# B&R Automation Studio project A65
Automation Studio 4.10.2.37

## Configuration Config1

CPU X20CP1382, AutomationRuntime D4.83, Build 4.1.2

### Task classes (Cpu.sw)
```
Cyclic#1 (cycle 2000 us, tolerance 2000 us):
  TaskFast <- Kontrol.TaskFast.TaskFast.prg
  FastMeter <- (binary)
  Program <- (binary)
  SslClient <- (binary)
  Server <- (binary)
  Client <- (binary)
  QDTA_IO <- (binary)
Cyclic#2 (cycle 10000 us, tolerance 10000 us):
  Protection <- Kontrol.Protection.Protection.prg
  Control <- Kontrol.Control.Control.prg
Cyclic#3 (cycle 100000 us, tolerance 100000 us):
  WatchDog <- WatchDog.WatchDog.prg
  System <- Kontrol.System.System.prg
  Hardware <- Kontrol.Hardware.Hardware.prg
  ProtUpdate <- Kontrol.Protection.ProtUpdate.prg
  Command <- Kontrol.Command.Command.prg
  cb52 <- Kontrol.CB52.cb52.prg
Cyclic#4 (cycle 200000 us, tolerance 200000 us):
  Auto <- Auto.Auto.prg
Cyclic#6 (cycle 50000 us, tolerance 3000000 us):
  MDB_Comand <- Auto.Modbus.MDB_Comando.prg
  MDB_Status <- Auto.Modbus.MDB_Status.prg
  MDB_Alarme <- Auto.Modbus.MDB_Alarme.prg
  MDB_Medida <- Auto.Modbus.MDB_Medida.prg
  MDB_Parame <- Auto.Modbus.MDB_Parametro.prg
Cyclic#7 (cycle 20000 us, tolerance 10000000 us):
  Event <- Kontrol.Event.Event.prg
  Comm <- Comm.Comm.prg
Cyclic#8 (cycle 50000 us, tolerance 10000000 us):
  File <- Kontrol.File.File.prg
Binaries: TCData, udbdef, ashwd, sysconf, asfw, arconfig, iomap, Role, User, ashwac, OpcUaMap, vccddbox, ihm01, ihm02, ihm03, vccpopup, vcpfx20, vcctrend, vccstr, vcmgr, vcpdsw, vcpdvnc, vccline, vccovl, arial, vcdsint, vccnum, vcalarm, vctcal, vccbtn, vcnet, vccbmp, vcrt, vcshared, vccdt, vcgclass, vcfntttf, vcbclass, vcdsloc, vcfile, arialbd, vcctext, vccshape, vccgauge, vcpkat, 10111548$f, Visu02, Visu03, Visu01, vccbar, vccslider, vcchspot, vccurl, vccalarm, vcchtml, vcxml
Libraries: operator, runtime, LoopConR, sys_lib, brsystem, AsTCP, AsIecCon, astime, AsBrStr, AsARCfg, AsXml, FileIO, AsIOAcc, standard, AsSem, IecCheck, DRV_mbus, dvframe, DataObj, Pgs0985, PgsAI4622, PgsAO4622, PgsAuto, PgsCfgNet, PgsComm, PgsControl, PgsEvent, PgsFileSys, PgsProt, PgsTag, PgsTagLink, PgsTelnet, vcresman, ashw
```

### Hardware
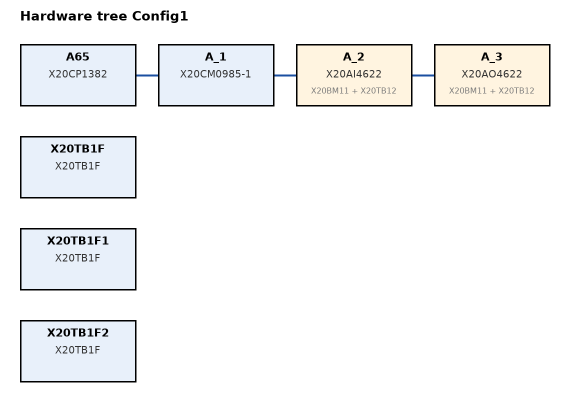
```
A65 : X20CP1382 v1.11.0.0  [X1 -> X1.SL; X2 -> X2.SL; X3 -> X3.SL]
  Module X1 (Type=X1, Virtual=true, Version=1.11.0.0)
    Connection (Connector=SS1, TargetModule=X20TB1F, TargetConnector=SS)
    Connection (Connector=SL, TargetModule=A65, TargetConnector=X1)
    X1AI_ChannelType01 = PT1000
    X1AI_ChannelType02 = 4 to 20mA
    X1AI2_LowerLimit_420mA = -8192
  Module X2 (Type=X2, Virtual=true, Version=1.11.0.0)
    Connection (Connector=SS1, TargetModule=X20TB1F1, TargetConnector=SS)
    Connection (Connector=SL, TargetModule=A65, TargetConnector=X2)
    X2CounterFunction = Edge
    X2CounterTimeInfo = 32Bit
  Module X3 (Type=X3, Virtual=true, Version=1.11.0.0)
    Connection (Connector=SS1, TargetModule=X20TB1F2, TargetConnector=SS)
    Connection (Connector=SL, TargetModule=A65, TargetConnector=X3)
  Connector IF1:
    Baudrate = 19200
  Connector IF2:
    ActivateDevice = 1
    Mode = Manual
    InternetAddress = 192.168.0.100
    SubnetMask = 255.255.255.0
    InaNodeNumber = 1
    Vnc1
    VncKeyMappingFile1 = 
    VncRefreshRate1 = 250
    ActivateSnmp = 2
    ActivateModbus = 1
    NumSlaves = -1
    NumAllBlocks = -1
    MemSizeIn = -1
    MemSizeOut = -1
  Connector IF3:
    DNAConfiguration = manual
    ActivateIna = 1
  ConfigurationID = A65
  RemanentGlobalPvSize = 10940
  EnableUsbRemoteInstall = 1
  EnableCfRemoteInstall = 1
  SystemTick = 2000
  IdleTaskClass = 8
  TaskClassIdleTime = 4000
  Cyclic1Duration = 2000
  Cyclic1Tolerance = 2000
  Cyclic2Duration = 10000
  Cyclic2Tolerance = 10000
  Cyclic3Duration = 100000
  Cyclic3Tolerance = 100000
  Cyclic4Duration = 200000
  Cyclic4Tolerance = 200000
  Cyclic5Duration = 500000
  Cyclic5Tolerance = 500000
  Cyclic6Duration = 50000
  Cyclic6Tolerance = 3000000
  Cyclic7Duration = 20000
  Cyclic7Tolerance = 10000000
  Cyclic8Duration = 50000
  Cyclic8Tolerance = 10000000
  FileDevice1
  FileDeviceName1 = 
  FileDevicePath1 = 
  TimeZone = 105
  ActivateSntp = 1
  SntpcServAddr1 = a.st1.ntp.br
  SntpcServAddr2 = b.st1.ntp.br
  SntpcServAddr3 = c.st1.ntp.br
  SntpcServAddr4 = d.st1.ntp.br
  EthernetDefaultGateway = 192.168.0.1
  FtpUser1
  FtpUsername1 = progressul
  FtpUserPassword1 = vk2iY3J4UkERtYbEJrmZIzULlFJLyE0YoKo7iPp2s1I=
  FtpUserSalt1 = 6vig95Eg
  FTPAccessRight1 = 0
  FTPMSPartition1 = SYSTEM
  FTPMSpath1 = 
  ActivateOpcUa = 1
  OpcUaInformationModels_PV_Version = 1
A_1 : X20CM0985-1 v2.2.0.0  [X2X1 -> A65.IF6]
  Supervision = off
  ReadBack = on
  FuncDO5 = NetErrorUser
  Timestamps = on
  GenErrorReset = on
  GenErrorCheck = phaseline
  NetConfig = 3Phase
  SyncConfig = X4X3
A_2 : X20AI4622 v1.1.0.0  [SS1 -> X20TB12.SS; SL -> X20BM11.SL1]
  Supervision = off
  ChannelType01 = 4 to 20mA
  ChannelType02 = 4 to 20mA
  ChannelType03 = 4 to 20mA
  ChannelType04 = 4 to 20mA
A_3 : X20AO4622 v1.2.0.0  [SS1 -> X20TB12j.SS; SL -> X20BM11i.SL1]
  Supervision = off
  ChannelType01 = 0 to 20mA
  ChannelType02 = 4 to 20mA
  ChannelType03 = 4 to 20mA
  ChannelType04 = 4 to 20mA
X20BM11 : X20BM11 v1.0.0.1  [X2X1 -> A_1.X2X2]
X20BM11i : X20BM11 v1.0.0.1  [X2X1 -> X20BM11.X2X2]
X20TB12 : X20TB12 v1.0.0.0
X20TB12j : X20TB12 v1.0.0.0
X20TB1F : X20TB1F v1.0.0.0
X20TB1F1 : X20TB1F v1.0.0.0
X20TB1F2 : X20TB1F v1.0.0.0
```

### IoMap.iom - A65/IoMap.iom
```iecst
(*********************************************************************************
 * Copyright: Microsoft
 * Author:    sandrionir
 * Created:   February 21, 2017/7:19 AM
 *********************************************************************************
 * IO mapping
 *********************************************************************************)
VAR_CONFIG
	Cyclic#4.HW.TemperatureENV AT %IW."A65".TemperatureENV;
	Cyclic#4.HW.TemperatureCPU AT %IW."A65".TemperatureCPU;
	Cyclic#2.cm0985IO.di.T32N AT %IX."A_1".StatusInput32;
	Cyclic#2.cm0985IO.di.T32P AT %IX."A_1".StatusInput31;
	Cyclic#2.cm0985IO.di.T27_2 AT %IX."A_1".StatusInput18;
	Cyclic#2.cm0985IO.di.T32Q AT %IX."A_1".StatusInput10;
	Cyclic#2.cm0985IO.di.T51 AT %IX."A_1".StatusInput09;
	Cyclic#2.cm0985IO.di.T50 AT %IX."A_1".StatusInput08;
	Cyclic#2.cm0985IO.di.T50N AT %IX."A_1".StatusInput07;
	Cyclic#2.cm0985IO.di.T60I AT %IX."A_1".StatusInput06;
	Cyclic#2.cm0985IO.di.T60V AT %IX."A_1".StatusInput05;
	Cyclic#2.cm0985IO.di.T81U AT %IX."A_1".StatusInput04;
	Cyclic#2.cm0985IO.di.T81O AT %IX."A_1".StatusInput03;
	Cyclic#2.cm0985IO.di.T27_1 AT %IX."A_1".StatusInput02;
	Cyclic#2.cm0985IO.di.T59 AT %IX."A_1".StatusInput01;
	Cyclic#2.::cm0985IO.do.RstError AT %QX."A_1".ResetGeneratorErrors;
	Cyclic#2.HW.Modulos.A_1_OK AT %IX."A_1".ModuleOk;
	Cyclic#2.cm0985IO.do.INVDO05 AT %QX."A_1".InvertDO5;
	Cyclic#2.Protection.do.trip_86h AT %QX."A_1".DigitalOutput06;
	Cyclic#2.Protection.do.trip_86e AT %QX."A_1".DigitalOutput05;
	Cyclic#2.::cm0985IO.do.SyncDeadBus AT %QX."A_1".ConfigOutput19;
	Cyclic#2.::cm0985IO.do.SyncCheck AT %QX."A_1".ConfigOutput18;
	Cyclic#2.::cm0985IO.do.SyncSlip AT %QX."A_1".ConfigOutput17;
	Cyclic#2.cm0985Meter.Registers.AnalogInput43 AT %ID."A_1".AnalogInput43;
	Cyclic#2.cm0985Meter.Registers.AnalogInput42 AT %ID."A_1".AnalogInput42;
	Cyclic#2.cm0985Meter.Registers.AnalogInput41 AT %ID."A_1".AnalogInput41;
	Cyclic#2.cm0985Meter.Registers.AnalogInput40 AT %ID."A_1".AnalogInput40;
	Cyclic#2.cm0985Meter.Registers.AnalogInput39 AT %ID."A_1".AnalogInput39;
	Cyclic#2.cm0985Meter.Registers.AnalogInput38 AT %ID."A_1".AnalogInput38;
	Cyclic#2.cm0985Meter.Registers.AnalogInput35 AT %IW."A_1".AnalogInput35;
	Cyclic#2.cm0985Meter.Registers.AnalogInput30 AT %IW."A_1".AnalogInput30;
	Cyclic#2.cm0985Meter.Registers.AnalogInput29 AT %IW."A_1".AnalogInput29;
	Cyclic#2.cm0985Meter.Registers.AnalogInput27 AT %IW."A_1".AnalogInput27;
	Cyclic#2.cm0985Meter.Registers.AnalogInput26 AT %IW."A_1".AnalogInput26;
	Cyclic#2.cm0985Meter.Registers.AnalogInput25 AT %IW."A_1".AnalogInput25;
	Cyclic#2.cm0985Meter.Registers.AnalogInput24 AT %IW."A_1".AnalogInput24;
	Cyclic#2.cm0985Meter.Registers.AnalogInput23 AT %IW."A_1".AnalogInput23;
	Cyclic#2.cm0985Meter.Registers.AnalogInput22 AT %IW."A_1".AnalogInput22;
	Cyclic#2.cm0985Meter.Registers.AnalogInput21 AT %IW."A_1".AnalogInput21;
	Cyclic#2.cm0985Meter.Registers.AnalogInput20 AT %IW."A_1".AnalogInput20;
	Cyclic#2.cm0985Meter.Registers.AnalogInput19 AT %IW."A_1".AnalogInput19;
	Cyclic#2.cm0985Meter.Registers.AnalogInput18 AT %IW."A_1".AnalogInput18;
	Cyclic#2.cm0985Meter.Registers.AnalogInput17 AT %IW."A_1".AnalogInput17;
	Cyclic#2.cm0985Meter.Registers.AnalogInput16 AT %IW."A_1".AnalogInput16;
	Cyclic#2.cm0985Meter.Registers.AnalogInput15 AT %IW."A_1".AnalogInput15;
	Cyclic#2.cm0985Meter.Registers.AnalogInput14 AT %IW."A_1".AnalogInput14;
	Cyclic#2.cm0985Meter.Registers.AnalogInput13 AT %IW."A_1".AnalogInput13;
	Cyclic#2.cm0985Meter.Registers.AnalogInput12 AT %IW."A_1".AnalogInput12;
	Cyclic#2.cm0985Meter.Registers.AnalogInput11 AT %IW."A_1".AnalogInput11;
	Cyclic#2.cm0985Meter.Registers.AnalogInput10 AT %IW."A_1".AnalogInput10;
	Cyclic#2.cm0985Meter.Registers.AnalogInput09 AT %IW."A_1".AnalogInput09;
	Cyclic#2.cm0985Meter.Registers.AnalogInput08 AT %IW."A_1".AnalogInput08;
	Cyclic#2.cm0985Meter.Registers.AnalogInput07 AT %IW."A_1".AnalogInput07;
	Cyclic#2.cm0985Meter.Registers.AnalogInput06 AT %IW."A_1".AnalogInput06;
	Cyclic#2.cm0985Meter.Registers.AnalogInput05 AT %IW."A_1".AnalogInput05;
	Cyclic#2.cm0985Meter.Registers.AnalogInput04 AT %IW."A_1".AnalogInput04;
	Cyclic#2.cm0985Meter.Registers.AnalogInput03 AT %IW."A_1".AnalogInput03;
	Cyclic#2.cm0985Meter.Registers.AnalogInput02 AT %IW."A_1".AnalogInput02;
	Cyclic#2.cm0985Meter.Registers.AnalogInput01 AT %IW."A_1".AnalogInput01;
	Cyclic#5.Control:rpm1.MasterCount AT %ID."X2".Counter01Value;
	Cyclic#5.Control:rpm1.MasterTime AT %ID."X2".Counter01TimeChanged;
	Cyclic#2.cm0985IO.di.UgPhSeqFault AT %IX."A_1".StatusInput19;
	Cyclic#2.cm0985IO.di.IgPhSeqFault AT %IX."A_1".StatusInput20;
	Cyclic#2.cm0985IO.di.UbPhSeqFault AT %IX."A_1".StatusInput21;
	Cyclic#2.cm0985IO.di.Us1PhSeqFault AT %IX."A_1".StatusInput22;
	Cyclic#2.::cm0985IO.di.PS24VFault AT %IX."A_1".StatusInput16;
	Cyclic#4.HW.SerialNumber AT %ID."A65".SerialNumber;
	Cyclic#4.HW.ModuleID AT %IW."A65".ModuleID;
	Cyclic#5.Control:rpm2.MasterCount AT %ID."X2".Counter02Value;
	Cyclic#5.Control:rpm2.MasterTime AT %ID."X2".Counter02TimeChanged;
	Cyclic#2.cm0985Meter.Registers.AnalogInput33 AT %IW."A_1".AnalogInput33;
	Cyclic#2.cm0985Meter.Registers.AnalogInput34 AT %IW."A_1".AnalogInput34;
	Cyclic#2.cm0985Meter.Registers.AnalogInput31 AT %IW."A_1".AnalogInput31;
	Cyclic#2.cm0985Meter.Registers.AnalogInput32 AT %IW."A_1".AnalogInput32;
	HW.FalhaFonteIO AT %IX."X3".StatusInput01;
	Protection.ai.ExcTemp AT %IW."X1".AnalogInput01;
	A65.ai.if AT %IW."X1".AnalogInput02;
	A65.di.dead_bus_enable AT %IX."X2".DigitalInput05;
	A65.di.avr_enable AT %IX."X2".DigitalInput01;
	A65.di.avr_ctrl_qm_enable AT %IX."X2".DigitalInput02;
	A65.di.avr_ctrl_pf_enable AT %IX."X2".DigitalInput03;
	A65.di.sync_enable AT %IX."X2".DigitalInput04;
	CB52.di.closed AT %IX."X2".DigitalInput06;
	A65.di.remote AT %IX."X2".DigitalInput07;
	A65.di.gov_trip AT %IX."X2".DigitalInput08;
	A65.di.avr_trip AT %IX."X2".DigitalInput09;
	A65.di.reset AT %IX."X1".DigitalInput01;
	A65.di.gov_enable AT %IX."X1".DigitalInput02;
	A65.di.gov_ctrl_pwr_enable AT %IX."X1".DigitalInput03;
	A65.di.gov_unload AT %IX."X1".DigitalInput04;
	A65.do.watchdog AT %QX."X3".DigitalOutput01;
	A65.do.gov_on AT %QX."X3".DigitalOutput02;
	A65.do.power_zero AT %QX."X3".DigitalOutput03;
	A65.ao.pwr AT %QW."A_3".AnalogOutput01;
	A65.ao.pos1 AT %QW."A_3".AnalogOutput02;
	Cyclic#4.HW.Modulos.A_3_OK AT %IX."A_3".ModuleOk;
	HW.Modulos.X1_Status AT %IB."X1".StatusInput01;
	A65.ao.pos2 AT %QW."A_3".AnalogOutput03;
	A65.ao.pos3 AT %QW."A_3".AnalogOutput04;
	Protection.di.crowbar_ok AT %IX."X2".DigitalInput10;
	Protection.di.pwr_temp_ok AT %IX."X2".DigitalInput14;
	A65.do.rotation_zero AT %QX."X3".DigitalOutput04;
	A65.do.rotation_nominal AT %QX."X3".DigitalOutput05;
	A65.do.rotation_brake AT %QX."X3".DigitalOutput06;
	A65.do.avr_on AT %QX."X3".DigitalOutput07;
	A65.do.field_flash_on AT %QX."X3".DigitalOutput08;
	A65.do.voltage_nominal AT %QX."X3".DigitalOutput09;
	A65.do.sync_enabled AT %QX."X3".DigitalOutput10;
	A65.do.dead_bus_enabled AT %QX."X3".DigitalOutput11;
	Protection.do.trip_50bf AT %QX."X3".DigitalOutput12;
	HW.Modulos.A_2_OK AT %IX."A_2".ModuleOk;
	A65.ai.uf AT %IW."A_2".AnalogInput01;
	A65.ai.pos1 AT %IW."A_2".AnalogInput02;
	A65.ai.pos2 AT %IW."A_2".AnalogInput03;
	A65.ai.pos3 AT %IW."A_2".AnalogInput04;
END_VAR
```

## Logical view

Binary libraries used (declarations not repeated): AsARCfg, AsBrStr, AsIecCon, AsIOAcc, AsSem, AsTCP, astime, AsXml, brsystem, DataObj, DRV_mbus, dvframe, FileIO, LoopConR 4.10.0, operator, runtime, standard, sys_lib, IecCheck, Pgs0985 2.00.0, PgsAI4622, PgsAO4622, PgsCfgNet, PgsComm 1.10.1, PgsControl, PgsEvent 1.00.0, PgsFileSys, PgsProt 2.00.0, PgsTag 2.02.0, PgsTagLink, PgsTelnet 2.01.1, MDB_Comando

### Global.typ - Global data types
```iecst
(*********************************************************************************
 * Copyright: Microsoft
 * Author:    sandrionir
 * Created:   February 21, 2017/7:19 AM
 *********************************************************************************
 * Global data types of project
 *********************************************************************************)

TYPE
	PgsVersionType : 	STRUCT
		X : UINT;
		Y : UINT;
		Z : UINT;
	END_STRUCT;
	PgsHW : 	STRUCT
		TemperatureCPU : UINT;
		TemperatureENV : UINT;
		SerialNumber : UDINT;
		ModuleID : UINT;
		FalhaFonteIO : BOOL;
		Modulos : PgsHWModulos;
	END_STRUCT;
	PgsHWModulos : 	STRUCT
		X1_Status : USINT;
		A_1_OK : BOOL;
		A_2_OK : BOOL;
		A_3_OK : BOOL;
		A_4_OK : BOOL;
		A_5_OK : BOOL;
		A_6_OK : BOOL;
		A_7_OK : BOOL;
		A_8_OK : BOOL;
		A_9_OK : BOOL;
		A_10_OK : BOOL;
		A_11_OK : BOOL;
		A_12_OK : BOOL;
	END_STRUCT;
END_TYPE
```

### Global.var - Global variables
```iecst
(*********************************************************************************
 * Copyright: Microsoft
 * Author:    sandrionir
 * Created:   February 21, 2017/7:19 AM
 *********************************************************************************
 * Global variables of project
 *********************************************************************************)
VAR CONSTANT
	version : PgsVersionType := (X:=2,Y:=2,Z:=0);
END_VAR
(*Hardware*)
VAR
	HW : PgsHW;
END_VAR
```

### Package Logical/Libraries - Global libraries

### Library Logical/Libraries/Kontrol/PgsAuto (IEC)
Depends on: sys_lib

#### PgsAuto.fun - Exported functions and function blocks
```iecst
FUNCTION_BLOCK PgsEnergia
	VAR_INPUT
		enable : BOOL;
		reset : BOOL;
		power : REAL;
		set_inicial : BOOL;
		set_posEnergy : REAL;
		set_negEnergy : REAL;
	END_VAR
	VAR_OUTPUT
		posEnergy : LREAL;
		negEnergy : LREAL;
	END_VAR
	VAR
		priv : PgsEnergiaPrivType;
	END_VAR
END_FUNCTION_BLOCK

FUNCTION_BLOCK PgsHorimetro
	VAR_INPUT
		enable : BOOL;
		reset : BOOL;
		set_inicial : BOOL;
		set_total : REAL;
	END_VAR
	VAR_OUTPUT
		total : REAL;
		horas : REAL;
		minutos : REAL;
		segundos : REAL;
	END_VAR
	VAR
		priv : PgsHorimetroPrivType;
	END_VAR
END_FUNCTION_BLOCK

FUNCTION_BLOCK PgsManobra
	VAR_INPUT
		enable : BOOL;
		reset : BOOL;
		set_inicial : BOOL;
		set_total : REAL;
	END_VAR
	VAR_OUTPUT
		total : REAL;
	END_VAR
	VAR
		priv : PgsManobraPrivType;
	END_VAR
END_FUNCTION_BLOCK

FUNCTION PGS_MDB_TO_REAL : REAL (*TODO: Add your comment here*) (*$GROUP=User,$CAT=User,$GROUPICON=User.png,$CATICON=User.png*)
	VAR_INPUT
		IN : UDINT;
	END_VAR
	VAR
		pVar : REFERENCE TO REAL;
		varUint : ARRAY[0..1] OF UINT;
		varUint1 : REFERENCE TO ARRAY[0..1] OF UINT;
	END_VAR
END_FUNCTION

FUNCTION PGS_REAL_TO_MDB : UDINT (*TODO: Add your comment here*) (*$GROUP=User,$CAT=User,$GROUPICON=User.png,$CATICON=User.png*)
	VAR_INPUT
		IN : REAL;
	END_VAR
	VAR
		pVar : REFERENCE TO UDINT;
		varUint : ARRAY[0..1] OF UINT;
		varUint1 : REFERENCE TO ARRAY[0..1] OF UINT;
	END_VAR
END_FUNCTION

{REDUND_ERROR} FUNCTION PGS_MDB_TO_DINT : DINT (*TODO: Add your comment here*) (*$GROUP=User,$CAT=User,$GROUPICON=User.png,$CATICON=User.png*)
	VAR_INPUT
		HIGH : UINT;
		LOW : UINT;
	END_VAR
	VAR
		pVar : REFERENCE TO DINT;
		varUint : ARRAY[0..1] OF UINT;
	END_VAR
END_FUNCTION

{REDUND_ERROR} FUNCTION PGS_MDB_TO_UDINT : UDINT (*TODO: Add your comment here*) (*$GROUP=User,$CAT=User,$GROUPICON=User.png,$CATICON=User.png*)
	VAR_INPUT
		HIGH : UINT;
		LOW : UINT;
	END_VAR
	VAR
		pVar : REFERENCE TO UDINT;
		varUint : ARRAY[0..1] OF UINT;
	END_VAR
END_FUNCTION

FUNCTION_BLOCK PgsAlarme
	VAR_INPUT
		IN : BOOL; (*input signal*)
		PT : TIME; (*delay time*)
		RESET : BOOL; (*resets output Q1*)
	END_VAR
	VAR_OUTPUT
		Q : BOOL; (*rising edge of the input signal is delayed by PT*)
	END_VAR
	VAR
		ton : TON;
	END_VAR
END_FUNCTION_BLOCK

{REDUND_ERROR} FUNCTION_BLOCK PgsFiltro (*TODO: Add your comment here*) (*$GROUP=User,$CAT=User,$GROUPICON=User.png,$CATICON=User.png*)
	VAR_INPUT
		IN : {REDUND_UNREPLICABLE} REAL;
		CTE : {REDUND_UNREPLICABLE} REAL;
	END_VAR
	VAR_OUTPUT
		OUT : {REDUND_UNREPLICABLE} REAL;
	END_VAR
	VAR
		acc : REAL;
	END_VAR
END_FUNCTION_BLOCK

{REDUND_ERROR} FUNCTION_BLOCK PgsEscala (*TODO: Add your comment here*) (*$GROUP=User,$CAT=User,$GROUPICON=User.png,$CATICON=User.png*)
	VAR_INPUT
		SensorMax : {REDUND_UNREPLICABLE} REAL;
		SensorMin : {REDUND_UNREPLICABLE} REAL;
		Entrada : REAL;
	END_VAR
	VAR_OUTPUT
		Valor : {REDUND_UNREPLICABLE} REAL;
		Sensor : REAL;
	END_VAR
	VAR
		filtro : PgsFiltro;
	END_VAR
END_FUNCTION_BLOCK

{REDUND_ERROR} FUNCTION_BLOCK PgsCabo (*TODO: Add your comment here*) (*$GROUP=User,$CAT=User,$GROUPICON=User.png,$CATICON=User.png*)
	VAR_INPUT
		IN : REAL;
		PT : TIME;
	END_VAR
	VAR_OUTPUT
		Falha : BOOL;
		Cabo_Aberto : BOOL;
		Cabo_Curto : BOOL;
	END_VAR
	VAR
		aberto : BOOL;
		curto : BOOL;
		ton_aberto : TON;
		ton_curto : TON;
	END_VAR
END_FUNCTION_BLOCK

{REDUND_OK} FUNCTION_BLOCK PgsSobre (*TODO: Add your comment here*) (*$GROUP=User,$CAT=User,$GROUPICON=User.png,$CATICON=User.png*)
	VAR_INPUT
		enable : BOOL := TRUE;
		IN : REAL;
		IN_AL : REAL;
		PT_AL : REAL;
		IN_TP : REAL;
		PT_TP : REAL;
		RST : BOOL;
	END_VAR
	VAR_OUTPUT
		Alarme : BOOL;
		Trip : BOOL;
	END_VAR
	VAR
		ton_al : TON;
		ton_tp : TON;
	END_VAR
END_FUNCTION_BLOCK

{REDUND_OK} FUNCTION_BLOCK PgsSub (*TODO: Add your comment here*) (*$GROUP=User,$CAT=User,$GROUPICON=User.png,$CATICON=User.png*)
	VAR_INPUT
		enable : BOOL := TRUE;
		IN : REAL;
		IN_AL : REAL;
		PT_AL : REAL;
		IN_TP : REAL;
		PT_TP : REAL;
		RST : BOOL;
	END_VAR
	VAR_OUTPUT
		Alarme : BOOL;
		Trip : BOOL;
	END_VAR
	VAR
		ton_al : TON;
		ton_tp : TON;
	END_VAR
END_FUNCTION_BLOCK

FUNCTION_BLOCK PgsX20AT
	VAR_INPUT
		Status : USINT;
	END_VAR
	VAR_OUTPUT
		IN1_Aberto : BOOL;
		IN1_Curto : BOOL;
		IN2_Aberto : BOOL;
		IN2_Curto : BOOL;
		IN3_Aberto : BOOL;
		IN3_Curto : BOOL;
		IN4_Aberto : BOOL;
		IN4_Curto : BOOL;
	END_VAR
END_FUNCTION_BLOCK

FUNCTION_BLOCK PgsStatusInput (*Para verificar o Status da Entrada Analógica*)
	VAR_INPUT
		Enable : BOOL;
		StatusInput : USINT; (*Status Input do módulo*)
		Pos : USINT; (*Posição da analógica 1,2,3 ou 4*)
		Reset : BOOL;
	END_VAR
	VAR_OUTPUT
		Limite_Inferior : BOOL;
		Limite_Superior : BOOL;
		Circuito_Aberto : BOOL;
	END_VAR
	VAR
		pos_0 : BOOL;
		pos_1 : BOOL;
	END_VAR
END_FUNCTION_BLOCK
```

#### PGS_MDB_TO_REAL.st
```iecst
(* TODO: Add your comment here *)
FUNCTION PGS_MDB_TO_REAL
    varUint1 ACCESS ADR(IN);
    varUint[0] := varUint1[1];
    varUint[1] := varUint1[0];
    pVar ACCESS ADR(varUint);
    PGS_MDB_TO_REAL := pVar;
END_FUNCTION
```

#### PGS_REAL_TO_MDB.st
```iecst
(* TODO: Add your comment here *)
FUNCTION PGS_REAL_TO_MDB
	varUint1 ACCESS ADR(IN);
    varUint[0] := varUint1[1];
    varUint[1] := varUint1[0];
    pVar ACCESS ADR(varUint);
    PGS_REAL_TO_MDB := pVar;
END_FUNCTION
```

#### PGS_MDB_TO_DINT.st
```iecst
(* TODO: Add your comment here *)
FUNCTION PGS_MDB_TO_DINT
    varUint[0] := HIGH;
    varUint[1] := LOW;
    pVar ACCESS ADR(varUint);
    PGS_MDB_TO_DINT := pVar;
END_FUNCTION
```

#### PgsAlarme.st
```iecst
(*<$Description$> TODO: Add your comment here </$Description$>*)
FUNCTION_BLOCK PgsAlarme

	ton(IN:=IN,PT:=PT);
	IF ton.Q  THEN
		Q	:= TRUE;
	ELSIF RESET THEN
		Q	:= FALSE;
	END_IF;

END_FUNCTION_BLOCK
```

#### PgsFiltro.st
```iecst
(* TODO: Add your comment here *)
FUNCTION_BLOCK PgsFiltro
	acc	:= acc + IN - OUT;
	OUT	:= acc / CTE;
END_FUNCTION_BLOCK
```

#### PgsEscala.st
```iecst
(* TODO: Add your comment here *)
FUNCTION_BLOCK PgsEscala

	Sensor	:= (Entrada / 32767.0) * 16.0 + 4.0;
	filtro(	IN:=((Sensor - 4.0) / 16.0)
				* (SensorMax - SensorMin)
				+  SensorMin,
			CTE:= 1);
	Valor   := filtro.OUT;

END_FUNCTION_BLOCK
```

#### PgsSobre.st
```iecst
(*<$Description$> TODO: Add your comment here </$Description$>*)
FUNCTION_BLOCK PgsSobre

	(* Alarme *)
	IF IN_AL = 0 THEN
		Alarme	:= FALSE;
	ELSE
		ton_al( IN := IN >= IN_AL , PT := REAL_TO_TIME( PT_AL * 1000) );
		IF ton_al.Q AND enable THEN
			Alarme	:= TRUE;
		ELSIF RST THEN
			Alarme	:= FALSE;
		END_IF;
	END_IF;

	(*Trip*)
	IF IN_TP = 0 THEN
		Trip	:= FALSE;
	ELSE
		ton_tp( IN := IN >= IN_TP , PT := REAL_TO_TIME( PT_TP * 1000) );
		IF ton_tp.Q AND enable THEN
			Trip	:= TRUE;
		ELSIF RST THEN
			Trip	:= FALSE;
		END_IF;
	END_IF;

END_FUNCTION_BLOCK
```

#### PgsEnergia.st
```iecst
(*<$Description$> TODO: Add your comment here </$Description$>*)
FUNCTION_BLOCK PgsEnergia

	priv.init_ton(IN:= priv.init, PT:=T#10s);
	IF priv.init_ton.Q THEN
		priv.init := FALSE;
		posEnergy := set_posEnergy;
		negEnergy := set_negEnergy;
	END_IF;

	priv.rt_info(enable := TRUE);
	priv.dh := UDINT_TO_REAL(priv.rt_info.cycle_time) / 3.6e9;

	IF enable THEN
		IF power > 0.0 THEN
			 posEnergy := posEnergy + power * priv.dh;
		ELSE
			 negEnergy := negEnergy + power * priv.dh;
		END_IF;
	END_IF;

	IF reset THEN
		reset := FALSE;
		posEnergy := 0.0;
		negEnergy := 0.0;
	END_IF;

	IF set_inicial THEN
		set_inicial := FALSE;
		posEnergy := set_posEnergy;
		negEnergy := set_negEnergy;
	END_IF;

	priv.bkp_ton(IN:= NOT priv.bkp_ton.Q, PT:=T#10m);
	IF priv.bkp_ton.Q THEN
		set_posEnergy := LREAL_TO_REAL(posEnergy);
		set_negEnergy := LREAL_TO_REAL(negEnergy);
	END_IF;
END_FUNCTION_BLOCK
```

#### PgsStatusInput.st
```iecst
(* TODO: Add your comment here *)
FUNCTION_BLOCK PgsStatusInput

IF Enable THEN

	CASE Pos OF
		1:	pos_0 := StatusInput.0;
			pos_1 := StatusInput.1;
		2:	pos_0 := StatusInput.2;
			pos_1 := StatusInput.3;
		3:	pos_0 := StatusInput.4;
			pos_1 := StatusInput.5;
		4:	pos_0 := StatusInput.6;
			pos_1 := StatusInput.7;
		ELSE
			pos_0 := TRUE;
			pos_1 := TRUE;
	END_CASE;

	IF pos_0 AND NOT pos_1  THEN
		Limite_Inferior := TRUE;
	ELSIF Reset THEN
		Limite_Inferior := FALSE;
	END_IF;
	IF NOT pos_0 AND pos_1  THEN
		Limite_Superior := TRUE;
	ELSIF Reset THEN
		Limite_Superior := FALSE;
	END_IF;
	IF pos_0 AND pos_1 THEN
		Circuito_Aberto := TRUE;
	ELSIF Reset THEN
		Circuito_Aberto := FALSE;
	END_IF;
ELSE
	Limite_Inferior := FALSE;
	Limite_Superior := FALSE;
	Circuito_Aberto := FALSE;
END_IF;

END_FUNCTION_BLOCK
```

### Program Logical/WatchDog/WatchDog (IEC)

#### Cyclic.st
```iecst
PROGRAM _CYCLIC
    License();
    ProtFlag.KeyInvalid			:= NOT License.Valid;
    ProtFlag.PwrSrcCpuIOFault	:= HW.FalhaFonteIO;
    ProtFlag.PwrSrcM1IOFault	:= cm0985IO.di.PS24VFault;

    IF  License.Valid                   AND
        NOT ProtFlag.PwrSrcCpuIOFault   AND	// Power Source CPU I/O Fault
        NOT ProtFlag.PwrSrcM1IOFault	AND // Power Source Energy Module I/O Fault
        HW.Modulos.A_1_OK				AND
        HW.Modulos.A_2_OK				AND
        HW.Modulos.A_3_OK		(*		AND
        HW.Modulos.A_4_OK				AND
        HW.Modulos.A_5_OK				AND
        HW.Modulos.A_6_OK				AND
        HW.Modulos.A_7_OK				AND
        HW.Modulos.A_8_OK				AND
        HW.Modulos.A_9_OK				AND
        HW.Modulos.A_10_OK				AND
        HW.Modulos.A_11_OK				AND
        HW.Modulos.A_12_OK		*)
        THEN
        WDOK    := TRUE;
    ELSE
        WDOK    := FALSE;
    END_IF

    //WatchDog
    ProtFlag.WatchDog	:= NOT WDOK;
	A65.do.watchdog		:= WDOK;

END_PROGRAM
```

### Share.typ
```iecst
TYPE
	PgsParEthType : 	STRUCT
		IF2_GATEWAY : STRING[16];
		IF2_BAUDRATE : USINT;
		IF2_MODE : USINT;
		IF2_IP : STRING[16];
		IF2_MASK : STRING[16];
		IF2_INA : USINT;
		IF3_MODE : USINT;
		IF3_IP : STRING[16];
		IF3_MASK : STRING[16];
		IF3_INA : USINT;
		update : BOOL;
		reading : BOOL;
		read_file : BOOL;
		write_file : BOOL;
	END_STRUCT;
END_TYPE
```

### Share.var
```iecst
(*Link Mobbus*)
VAR
	link_avr : PgsMbLinkAvrOpen;
	link_gov : PgsMbLinkGovOpen;
	link_pos1 : PgsMbLinkPosOpen;
	link_pos2 : PgsMbLinkPosOpen;
	link_pos3 : PgsMbLinkPosOpen;
	link_curve1 : PgsMbLinkCurveOpen;
	link_curve2 : PgsMbLinkCurveOpen;
	link_curve3 : PgsMbLinkCurveOpen;
	link_meter : PgsMbLinkRealOpen;
	link_system : PgsMbLinkRealOpen;
	link_sysIO : PgsMbLinkRealOpen;
	link_prot : PgsMbLinkRealOpen;
	link_mdb_medidas : PgsMbLinkRealOpen;
	link_mdb_parametros : PgsMbLinkRealOpen;
END_VAR
```

### Program Logical/Comm/Comm

#### Variables.var
```iecst
VAR
	mbusData : PgsMbDataOpen;
	mbusDevice : PgsMbDevice;
	mbusSetBlock : PgsMbSetBlock;
	mbusSetLink : PgsMbSetLink;
	mbusDataClose : PgsMbDataClose;
	mbusLinkClose : PgsMbLinkClose;
	mbusTcpOpen : PgsMbTcpOpen;
	mbusTcpUpdate : PgsMbTcpUpdate;
	mbusTcpClose : PgsMbTcpClose;
	telnetOpen : PgsTelnetOpen;
	telnetUpdate : PgsTelnetUpdate;
	telnetClose : PgsTelnetClose;
END_VAR
```

#### Cyclic.st
```iecst
PROGRAM _CYCLIC

    IF NOT PgsTagValid(TagManager.ident) THEN
        RETURN;
    END_IF

    mbusTcpUpdate   ( ident := mbusTcpOpen.ident );
    telnetUpdate(
        ident       := telnetOpen.ident,
        tagIdent    := TagManager.ident,
        evtIdent    := Event
    );

END_PROGRAM
```

#### Exit.st
```iecst
PROGRAM _EXIT

	mbusDataClose( dtaIdent := mbusData.dtaIdent );

	mbusLinkClose( lnkIdent := link_avr.Ident );
	mbusLinkClose( lnkIdent := link_gov.Ident );

	mbusLinkClose( lnkIdent := link_pos1.Ident );
	mbusLinkClose( lnkIdent := link_pos2.Ident );
	mbusLinkClose( lnkIdent := link_pos3.Ident );
	mbusLinkClose( lnkIdent := link_curve1.Ident );
	mbusLinkClose( lnkIdent := link_curve2.Ident );
	mbusLinkClose( lnkIdent := link_curve3.Ident );

	mbusLinkClose( lnkIdent := link_meter.Ident );

	mbusLinkClose( lnkIdent := link_system.Ident );
	mbusLinkClose( lnkIdent := link_sysIO.Ident );
	mbusLinkClose( lnkIdent := link_prot.Ident );

	mbusLinkClose( lnkIdent := link_mdb_medidas.Ident );
	mbusLinkClose( lnkIdent := link_mdb_parametros.Ident );

    mbusTcpClose( enable := TRUE, ident := mbusTcpOpen.ident );

    telnetClose( enable := TRUE, ident := telnetOpen.ident );

END_PROGRAM
```

#### Init.st
```iecst
PROGRAM _INIT

    mbusData( Devices := 1 );

	//Device 1
    mbusDevice(
        dtaIdent        := mbusData.dtaIdent,
        id              := 1,
		Links			:= 6,
		InputBlocks		:= 1,
        CoilBlocks      := 3
    );

    //AVR
	link_avr(
		CoilAddress		:= 4097,
		HoldingAddress	:= 5121,
		InputAddress	:= 7169,
        //GainUm          := 10.0,
        //GainIm          := 10.0,
        //GainSm          := 10.0,
        //GainUf          := 100.0,
        //GainIf          := 100.0,
		Float			:= TRUE,
		ModiconFormat	:= TRUE
	);
	mbusSetLink(
		devIdent	:= mbusDevice.devIdent,
		lnkIdent	:= link_avr.Ident
	);

    //GOV
	link_gov(
		CoilAddress		:= 8193,
		HoldingAddress	:= 9217,
		InputAddress	:= 11265,
        //GainUm          := 10.0,
        //GainSm          := 10.0,
		Float			:= TRUE,
		ModiconFormat	:= TRUE
	);
	mbusSetLink(
		devIdent	:= mbusDevice.devIdent,
		lnkIdent	:= link_gov.Ident
	);

	//POS1
	link_pos1(
		CoilAddress		:= 12289,
		HoldingAddress	:= 12545,
		InputAddress	:= 13569,
		Float			:= TRUE,
		ModiconFormat	:= TRUE
	);
	mbusSetLink(
		devIdent	:= mbusDevice.devIdent,
		lnkIdent	:= link_pos1.Ident
	);
	//Curve1
	link_curve1(
		HoldingAddress	:= 13825,
		InputAddress	:= 13953,
		Float			:= TRUE,
		ModiconFormat	:= TRUE
	);
	mbusSetLink(
		devIdent	:= mbusDevice.devIdent,
		lnkIdent	:= link_curve1.Ident
	);

	//POS2
	link_pos2(
		CoilAddress		:= 14337,
		HoldingAddress	:= 14593,
		InputAddress	:= 15617,
		Float			:= TRUE,
		ModiconFormat	:= TRUE
	);
	mbusSetLink(
		devIdent	:= mbusDevice.devIdent,
		lnkIdent	:= link_pos2.Ident
	);
	//Curve2
	link_curve2(
		HoldingAddress	:= 15873,
		InputAddress	:= 16001,
		Float			:= TRUE,
		ModiconFormat	:= TRUE
	);
	mbusSetLink(
		devIdent	:= mbusDevice.devIdent,
		lnkIdent	:= link_curve2.Ident
	);

	//POS3
	link_pos3(
		CoilAddress		:= 16385,
		HoldingAddress	:= 16641,
		InputAddress	:= 17665,
		Float			:= TRUE,
		ModiconFormat	:= TRUE
	);
	mbusSetLink(
		devIdent	:= mbusDevice.devIdent,
		lnkIdent	:= link_pos3.Ident
	);
	//Curve3
	link_curve3(
		HoldingAddress	:= 17921,
		InputAddress	:= 18049,
		Float			:= TRUE,
		ModiconFormat	:= TRUE
	);
	mbusSetLink(
		devIdent	:= mbusDevice.devIdent,
		lnkIdent	:= link_curve3.Ident
	);

    // MdbMeter
	link_meter(
        pBlock	        := ADR(MdbMeter),
        blockLen	    := SIZEOF(MdbMeter),
		Address			:= 2561,
		Holding			:= FALSE,
		//Gain			:= 10.0,
		Float			:= TRUE,
		ModiconFormat	:= TRUE
	);
	mbusSetLink(
		devIdent	:= mbusDevice.devIdent,
		lnkIdent	:= link_meter.Ident
	);

    // System Parameter
	link_system(
        pBlock	        := ADR(SysPar),
        blockLen	    := SIZEOF(SysPar),
		Address			:= 1025,
		Holding			:= TRUE,
		//Gain			:= 10,
		Float			:= TRUE,
		ModiconFormat	:= TRUE
	);
	mbusSetLink(
		devIdent	:= mbusDevice.devIdent,
		lnkIdent	:= link_system.Ident
	);
    //
    link_sysIO(
        pBlock	        := ADR(SysIOPar),
        blockLen	    := SIZEOF(SysIOPar),
		Address			:= 1255,
		Holding			:= TRUE,
		//Gain			:= 10,
		Float			:= TRUE,
		ModiconFormat	:= TRUE
	);
	mbusSetLink(
		devIdent	:= mbusDevice.devIdent,
		lnkIdent	:= link_sysIO.Ident
	);

    //SysUpdate
 	mbusSetBlock(
        devIdent    := mbusDevice.devIdent,
        BlockType   := PGS_MB_BLK_COIL,
        Address     := 1,
        pBlock      := ADR(SysUpdate),
        blockLen    := SIZEOF(SysUpdate)
    );

    //Protections
 	mbusSetBlock(
        devIdent    := mbusDevice.devIdent,
        BlockType   := PGS_MB_BLK_COIL,
        Address     := 40961,
        pBlock      := ADR(ProtFlag),
        blockLen    := SIZEOF(ProtFlag)
	);
	// Protections Parameter
	link_prot(
		pBlock	        := ADR(ProtPar),
		blockLen	    := SIZEOF(ProtPar),
		Address			:= 41985,
		Holding			:= TRUE,
		//Gain			:= 10,
		Float			:= TRUE,
		ModiconFormat	:= TRUE
	);
	mbusSetLink(
		devIdent	:= mbusDevice.devIdent,
		lnkIdent	:= link_prot.Ident
	);

//==================================================================================================================
    //Automação
    link_mdb_medidas(
		pBlock	        := ADR(MDB_Medidas),
		blockLen	    := SIZEOF(MDB_Medidas),
		Address			:= 20000,
		Holding			:= FALSE,
		//Gain			:= 10,
		Float			:= TRUE,
		ModiconFormat	:= TRUE
	);
	mbusSetLink(
		devIdent	:= mbusDevice.devIdent,
		lnkIdent	:= link_mdb_medidas.Ident
	);
    link_mdb_parametros(
		pBlock	        := ADR(MDB_Parametros),
		blockLen	    := SIZEOF(MDB_Parametros),
		Address			:= 21000,
		Holding			:= TRUE,
		//Gain			:= 10,
		Float			:= TRUE,
		ModiconFormat	:= TRUE
	);
	mbusSetLink(
		devIdent	:= mbusDevice.devIdent,
		lnkIdent	:= link_mdb_parametros.Ident
	);
	mbusSetBlock(
        devIdent    := mbusDevice.devIdent,
        BlockType   := PGS_MB_BLK_COIL,
        Address     := 22000,
        pBlock      := ADR(MDB_Status),
        blockLen    := SIZEOF(MDB_Status)
    );
	mbusSetBlock(
        devIdent    := mbusDevice.devIdent,
        BlockType   := PGS_MB_BLK_COIL,
        Address     := 23000,
        pBlock      := ADR(MDB_Comandos),
        blockLen    := SIZEOF(MDB_Comandos)
    );
	mbusSetBlock(
		devIdent    := mbusDevice.devIdent,
		BlockType   := PGS_MB_BLK_COIL,
		Address     := 24000,
		pBlock      := ADR(MDB_Alarmes),
		blockLen    := SIZEOF(MDB_Alarmes)
    );

//==================================================================================================================

    //TCP
    mbusTcpOpen (
        enable      := TRUE,
        dtaIdent    := mbusData.dtaIdent,
        port        := 502
    );
    mbusTcpUpdate.enable    := TRUE;
    mbusTcpUpdate.timeout   := 5.0;

    //Telnet
    telnetOpen (
        enable      := TRUE,
        port        := 23
    );
    telnetUpdate.enable    := TRUE;
    telnetUpdate.timeout   := 3600.0;

END_PROGRAM
```

### Program Logical/Kontrol/TaskFast/TaskFast (IEC)

#### Variables.var
```iecst
VAR
	uf_filter : PgsFiltro;
	if_filter : PgsFiltro;
END_VAR
```

#### Cyclic.st
```iecst
PROGRAM _CYCLIC

    //Uf : Field Voltage
    uf_filter( IN := INT_TO_REAL(A65.ai.uf) );
    UfAvg   := uf_filter.OUT;
    //If : Field Voltage
    if_filter( IN := INT_TO_REAL(A65.ai.if) );
    IfAvg   := if_filter.OUT;

END_PROGRAM
```

#### Init.st
```iecst
PROGRAM _INIT

	//Filters
    uf_filter.CTE      := 32;
    if_filter.CTE      := 32;

END_PROGRAM
```

### Share.typ
```iecst
TYPE
	PgsCM0985di : 	STRUCT
		PS24VFault : BOOL;
		UgPhSeqFault : BOOL;
		IgPhSeqFault : BOOL;
		UbPhSeqFault : BOOL;
		Us1PhSeqFault : BOOL;
		Us2PhSeqFault : BOOL;
		T59 : BOOL;
		T27_1 : BOOL;
		T27_2 : BOOL;
		T81O : BOOL;
		T81U : BOOL;
		T60V : BOOL;
		T60I : BOOL;
		T50N : BOOL;
		T50 : BOOL;
		T51 : BOOL;
		T32Q : BOOL;
		T32P : BOOL;
		T32N : BOOL;
		FO01 : BOOL;
		FO02 : BOOL;
		FO03 : BOOL;
		FO04 : BOOL;
		FO05 : BOOL;
		FO06 : BOOL;
	END_STRUCT;
	PgsCM0985do : 	STRUCT
		INVDO05 : BOOL;
		RstError : BOOL;
		SyncSlip : BOOL;
		SyncCheck : BOOL;
		SyncDeadBus : BOOL;
	END_STRUCT;
	PgsCM0985io : 	STRUCT
		di : PgsCM0985di;
		do : PgsCM0985do;
	END_STRUCT;
END_TYPE
```

### Share.var
```iecst
VAR
	CfgNet : PgsCfgNet := (parameter:=(if2:=(HostName:='Kontroll',baudrate:=PGS_CFG_NET_BAUDRATE_AUTO,mode:=PGS_CFG_NET_MODE_MANUAL,gateway:='192.168.0.1',ip:='192.168.0.100',mask:='255.255.255.0',ina:=1),if3:=(mode:=PGS_CFG_NET_MODE_MANUAL,ip:='10.0.0.100',mask:='255.0.0.0',ina:=2),ntp:=(timezone:=UTC03N,serverAddr1:='200.160.7.186',serverAddr2:='201.49.148.135',serverAddr3:='200.186.125.195',serverAddr4:='200.20.186.76')));
END_VAR
(*X20CM0985-1*)
VAR
	cm0985IO : PgsCM0985io;
	cm0985 : Pgs0985 := (Fnom:=60.0,EnableSetDO5:=TRUE,EnableSetDO6:=TRUE,ClockWise:=TRUE);
	cm0985DO1 : Pgs0985DO1 := (ResetManual:=FALSE,T59_1:=FALSE,T59_2:=FALSE,T27_1:=FALSE,T27_2:=FALSE,T81O_1:=FALSE,T81O_2:=FALSE,T81U_1:=FALSE,T81U_2:=FALSE,T60V:=FALSE,T60I:=FALSE,T50N:=FALSE,T50:=FALSE,T51:=FALSE,T32Q:=FALSE,T32P:=FALSE,T32N:=FALSE);
	cm0985Main : Pgs0985Main := (Enable3phase:=FALSE,Connection1:=PGS_0985_CON_ABC,V1prim:=115,V1sec:=115,V1nom:=115,Connection2:=PGS_0985_CON_ABCN,V2prim:=115,V2sec:=115,V2nom:=115);
	cm0985Bus : Pgs0985Bus := (Connection:=PGS_0985_CON_ABC,Vprim:=115,Vsec:=115,Vnom:=115);
	cm0985Sync : Pgs0985Sync := (Mode:=PGS_0985_SYNC_X4_X3,ChangeDO4toDo6:=FALSE,dFmax:=0.3,dFmin:=-0.3,dUmax:=10,dAngleMax:=5,PhaseShift:=0,UBmin:=0.05,DO4Pulse:=1,DO4SwTime:=0.1,DO6Pulse:=1,DO6SwTime:=0.1);
	cm0985Meter : Pgs0985Meter;
	cm0985Gen : Pgs0985Gen := (Connection:=PGS_0985_CON_ABCN,Vprim:=115,Vsec:=115,Vnom:=115,Iprim:=5,Isec:=5,Inom:=5,EnableHarmonic:=FALSE,Tfilter:=100,D02Pulse:=1);
	cm0985GenPu : Pgs0985GenPu;
	cm0985GenPf : Pgs0985GenPf;
	cm0985GenPa : Pgs0985GenPa;
	cm0985GenPc : Pgs0985GenPc;
	cm0985GenPp : Pgs0985GenPp;
	cm0985Update : Pgs0985Update;
END_VAR
(*X20AO4622*)
VAR
	ao4622 : PgsAO4622 := (Channel1:=PGS_AO4622_4_20_mA,Channel2:=PGS_AO4622_0_20_mA,Channel3:=PGS_AO4622_0_20_mA,Channel4:=PGS_AO4622_0_20_mA); (*ao4622Update : PgsAO4622Update;*)
END_VAR
(*X20AI4622*)
VAR
	ai4622 : PgsAI4622 := (FilterLevel:=PGS_AI4622_FILTER_LEVEL_002,RampLimit:=PGS_AI4622_RAMP_255,UpperLimit:=32767,LowerLimit:=-32768,Channel1:=PGS_AI4622_0_20_mA,Channel2:=PGS_AI4622_0_20_mA,Channel3:=PGS_AI4622_0_20_mA,Channel4:=PGS_AI4622_0_20_mA); (*ai4622Update : PgsAI4622Update;*)
END_VAR
```

### Program Logical/Kontrol/Hardware/Hardware (IEC)

#### Variables.var
```iecst
VAR
	Update0985 : BOOL; (*UpdateAI4622 : BOOL;
	UpdateAO4622 : BOOL;*)
	reset_cfg_net : TON;
END_VAR
```

#### Cyclic.st
```iecst
PROGRAM _CYCLIC

    CfgNet();

	reset_cfg_net(IN:=A65.di.reset, PT:=T#30s);

    // Check Reset Input
	IF reset_cfg_net.Q THEN
		CfgNet.parameter.if2.HostName	:= 'Kontroll';
		CfgNet.parameter.if2.ip			:= '192.168.000.100';
		CfgNet.parameter.if2.mask		:= '255.255.255.000';
		CfgNet.parameter.if2.gateway	:= '192.168.000.001';
		CfgNet.parameter.if2.baudrate	:= PGS_CFG_NET_BAUDRATE_AUTO;
		CfgNet.parameter.if2.mode		:= PGS_CFG_NET_MODE_MANUAL;
		CfgNet.parameter.if2.ina		:= 1;
		CfgNet.set  := TRUE;
	END_IF;

	IF PgsTagValid(TagManager.ident) AND Update0985 THEN
		Update0985 := FALSE;
        cm0985();
		cm0985Gen();
		cm0985Main();
		cm0985Bus();
		cm0985GenPu();
        cm0985GenPf();
        cm0985GenPa();
        cm0985GenPc();
        cm0985GenPp();
		cm0985DO1();
        cm0985Sync();
	END_IF
    cm0985Update();

END_PROGRAM
```

### Program Logical/Kontrol/System/System (IEC)

#### Cyclic.st
```iecst
PROGRAM _CYCLIC

	IF SysUpdate.SaveAll THEN
		SysUpdate.SaveAll		:= FALSE;
		SysUpdate.UpdateAll     := TRUE;
		TagUpdate.write         := TRUE;
	END_IF;

	IF PgsTagValid(TagManager.ident) AND SysUpdate.UpdateAll THEN
		SysUpdate.UpdateAll		:= FALSE;
		SysUpdate.UpdateGen		:= TRUE;
		SysUpdate.UpdateSync	:= TRUE;
		SysUpdate.UpdateBus		:= TRUE;
		SysUpdate.UpdateProt	:= TRUE;
		SysUpdate.UpdateIO      := TRUE;

		avr.Update				:= TRUE;
		gov.Update				:= TRUE;
		pos1.Update				:= TRUE;
		pos2.Update				:= TRUE;
		pos3.Update				:= TRUE;
	END_IF;

	IF SysUpdate.UpdateGen THEN
		SysUpdate.UpdateGen         := FALSE;
		SysUpdate.UpdateProt		:= TRUE;

		//Meter Base
		meter.Base.Um               := SysPar.Gen.UmNom;
		meter.Base.Sm               := SysPar.Gen.SmNom;
		meter.Base.Rot              := SysPar.Gen.RpmNom;
		meter.Base.Fm               := SysPar.Gen.FmNom;
		meter.Base.Uf               := SysPar.Gen.UfNom;
		meter.Base.If               := SysPar.Gen.IfNom;
		meter();

        //Phase Sequence
        cm0985.ClockWise            := REAL_TO_BOOL(SysPar.Gen.ClockWise);
        cm0985();

        //CM0985 - X2 and X3 - Generator
        cm0985Gen.Connection        := REAL_TO_UDINT(SysPar.Gen.Connection);
		cm0985Gen.Vprim             := SysPar.Gen.UmPrim;
		cm0985Gen.Vsec	            := SysPar.Gen.UmSec;
		cm0985Gen.Vnom		        := meter.Base.Um;
		cm0985Gen.Iprim		        := SysPar.Gen.ImPrim;
		cm0985Gen.Isec		        := REAL_TO_USINT(SysPar.Gen.ImSec);
		cm0985Gen.Inom		        := meter.Base.Im;
		cm0985Gen();
	END_IF;

	IF SysUpdate.UpdateSync THEN
		SysUpdate.UpdateSync        := FALSE;

        //Meter Base
        meter.Base.Ub               := SysPar.Sync.U1Nom;
		//CM0985 - X4 and X6 - Main
		//X4
        cm0985Main.Enable3phase     := REAL_TO_BOOL(SysPar.Sync.Enable3Phase);
        cm0985Main.Connection1      := REAL_TO_UDINT(SysPar.Sync.Connection);
		cm0985Main.V1prim			:= SysPar.Sync.U1Prim;
		cm0985Main.V1sec			:= SysPar.Sync.U1Sec;
		cm0985Main.V1nom			:= SysPar.Sync.U1Nom;
		cm0985Main();

		//CM0985 - Sync
		cm0985Sync.dFmax			:= SysPar.Sync.dFmax;
		cm0985Sync.dFmin			:= SysPar.Sync.dFmin;
		cm0985Sync.dUmax			:= SysPar.Sync.dUmax;
        cm0985Sync.UBmin            := SysPar.Sync.UBmin;
		cm0985Sync.dAngleMax		:= SysPar.Sync.dAngleMax;
		cm0985Sync.PhaseShift		:= SysPar.Sync.PhaseShift;
		cm0985Sync();

	END_IF;

	IF SysUpdate.UpdateBus THEN
		SysUpdate.UpdateBus         := FALSE;
		//CM0985 - X5 - Bus
		cm0985Bus.Vprim				:= SysPar.Exc.UexcPrim;
		cm0985Bus.Vsec				:= SysPar.Exc.UexcSec;
		cm0985Bus.Vnom				:= SysPar.Exc.UexcSec;
		cm0985Bus();
	END_IF;

	IF SysUpdate.ResetRunningHourMeter THEN
		SysUpdate.ResetRunningHourMeter	:= FALSE;
		hour_running.reset				:= TRUE;
	END_IF;

	IF SysUpdate.ResetOnlineHourMeter THEN
		SysUpdate.ResetOnlineHourMeter	:= FALSE;
		hour_online.reset				:= TRUE;
	END_IF;

//	IF SysUpdate.ResetEnergy THEN
//		SysUpdate.ResetEnergy			:= FALSE;
//		energia_ativa.reset				:= TRUE;
//		energia_reativa.reset			:= TRUE;
//	END_IF;

	IF SysUpdate.ResetEnergy THEN
		SysUpdate.ResetEnergy			:= FALSE;
		energy_active.reset				:= TRUE;
		energy_reactive.reset			:= TRUE;
	END_IF;

    IF SysUpdate.UpdateIO THEN
		SysUpdate.UpdateIO          := FALSE;

        //AI4622
        ai4622.Channel1             := REAL_TO_UDINT(SysIOPar.AI1Type);
        ai4622.Channel2             := REAL_TO_UDINT(SysIOPar.AI2Type);
        ai4622.Channel3             := REAL_TO_UDINT(SysIOPar.AI3Type);
        ai4622.Channel4             := REAL_TO_UDINT(SysIOPar.AI4Type);
        ai4622();

        //AO4622
        ao4622.Channel1             := REAL_TO_UDINT(SysIOPar.AO1Type);
        ao4622.Channel2             := REAL_TO_UDINT(SysIOPar.AO2Type);
        ao4622.Channel3             := REAL_TO_UDINT(SysIOPar.AO3Type);
        ao4622.Channel4             := REAL_TO_UDINT(SysIOPar.AO4Type);
	    ao4622();
	END_IF;

(****************** Hour Meter  ***********************)
	hour_running	( enable := meter.Out.Rot > 0.0 );
	hour_online		( enable := CB52.st.closed );

(***************** Energy Meter  **********************)
//	energia_ativa	( enable	:= CB52.st.closed,
//					  power		:= meter.In.Pm	);
//	energia_reativa	( enable	:= CB52.st.closed,
//					  power		:= meter.In.Qm	);

	// Update Meters
	MdbMeter[0]	 	:= meter.In.Fm;
	MdbMeter[1]	 	:= cm0985Meter.Ug1;
	MdbMeter[2]	 	:= cm0985Meter.Ug2;
	MdbMeter[3]	 	:= cm0985Meter.Ug3;
	MdbMeter[4]	 	:= cm0985Meter.Ug12;
	MdbMeter[5]	 	:= cm0985Meter.Ug23;
	MdbMeter[6]	 	:= cm0985Meter.Ug31;
	MdbMeter[7]	 	:= cm0985Meter.Ug;
	IF cm0985Meter.Ig > 5 THEN
		MdbMeter[8]	 	:= cm0985Meter.Ig1;
		MdbMeter[9]		:= cm0985Meter.Ig2;
		MdbMeter[10] 	:= cm0985Meter.Ig3;
		MdbMeter[11] 	:= cm0985Meter.Ig;
	ELSE
		MdbMeter[8]	 	:= 0;
		MdbMeter[9]		:= 0;
		MdbMeter[10] 	:= 0;
		MdbMeter[11] 	:= 0;
	END_IF;

	MdbMeter[12] 	:= cm0985Meter.Ign;
	MdbMeter[13] 	:= cm0985Meter.Igm_dyn;
	MdbMeter[14] 	:= cm0985Meter.Pg;
	MdbMeter[15] 	:= cm0985Meter.Qg;
	MdbMeter[16] 	:= cm0985Meter.Sg;
	MdbMeter[17] 	:= meter.In.PF;
    //Exc
	MdbMeter[18]    := uf_input;
	MdbMeter[19] 	:= filter_uf.y; //meter.In.Uf;
	MdbMeter[20]    := if_input;
	MdbMeter[21] 	:= meter.In.If;
	MdbMeter[22] 	:= cm0985Meter.Fb;
	MdbMeter[23] 	:= cm0985Meter.Ub12;
	MdbMeter[24] 	:= cm0985Meter.Ub23;
	MdbMeter[25] 	:= cm0985Meter.Ub31;
    //Bus
	MdbMeter[26] 	:= cm0985Meter.Un1;
	MdbMeter[27] 	:= cm0985Meter.Un2;
	MdbMeter[28] 	:= cm0985Meter.Un3;
	MdbMeter[29] 	:= cm0985Meter.Un12;
	MdbMeter[30] 	:= cm0985Meter.Un23;
	MdbMeter[31] 	:= cm0985Meter.Un31;
	MdbMeter[32] 	:= cm0985Meter.Fs1;
	IF cm0985Meter.dAngle > 180 THEN
		MdbMeter[33]:= cm0985Meter.dAngle - 360;
	ELSE
		MdbMeter[33]:= cm0985Meter.dAngle;
	END_IF
    //Turbine
	MdbMeter[34] 	:= meter.In.Rot;
	MdbMeter[35] 	:= pos1_input;
	MdbMeter[36] 	:= pos1.PosIn;
	MdbMeter[37] 	:= pos2_input;
	MdbMeter[38] 	:= pos2.PosIn;
	MdbMeter[39] 	:= pos3_input;
	MdbMeter[40] 	:= pos3.PosIn;
    //
	MdbMeter[41] 	:= ExcTemp;												//Excitation Temperature
	MdbMeter[42]	:= hour_running.horas;
	MdbMeter[43]	:= hour_running.minutos;
	MdbMeter[44]	:= hour_online.horas;
	MdbMeter[45]	:= hour_online.minutos;
	MdbMeter[46]	:= LREAL_TO_REAL(energy_active.posEnergy); //LREAL_TO_REAL(energia_ativa.posEnergy);
	MdbMeter[47]	:= LREAL_TO_REAL(energy_active.negEnergy); //LREAL_TO_REAL(energia_ativa.negEnergy);
	MdbMeter[48]	:= LREAL_TO_REAL(energy_reactive.posEnergy); //LREAL_TO_REAL(energia_reativa.posEnergy);
	MdbMeter[49]	:= LREAL_TO_REAL(energy_reactive.negEnergy); //LREAL_TO_REAL(energia_reativa.negEnergy);

END_PROGRAM
```

#### Init.st
```iecst
PROGRAM _INIT
    TagManager(enable:=TRUE);
    //Register Parameters
    PgsTagStartNode     (TagManager.ident, ADR('system'));
    //Sync
    PgsTagStartNode     (TagManager.ident, ADR('sync'));
    PgsTagRegisterREAL  (TagManager.ident, TRUE, ADR('U1Prim'),         SysPar.Sync.U1Prim);
    PgsTagRegisterREAL  (TagManager.ident, TRUE, ADR('U1Sec'),          SysPar.Sync.U1Sec);
    PgsTagRegisterREAL  (TagManager.ident, TRUE, ADR('Enable3Phase'),   SysPar.Sync.Enable3Phase);
    PgsTagRegisterREAL  (TagManager.ident, TRUE, ADR('Connection'),     SysPar.Sync.Connection);
    PgsTagRegisterREAL  (TagManager.ident, TRUE, ADR('U1Nom'),          SysPar.Sync.U1Nom);
    PgsTagRegisterREAL  (TagManager.ident, TRUE, ADR('UBmin'),          SysPar.Sync.UBmin);
    PgsTagRegisterREAL  (TagManager.ident, TRUE, ADR('dFmax'),          SysPar.Sync.dFmax);
    PgsTagRegisterREAL  (TagManager.ident, TRUE, ADR('dFmin'),          SysPar.Sync.dFmin);
    PgsTagRegisterREAL  (TagManager.ident, TRUE, ADR('dUmax'),          SysPar.Sync.dUmax);
    PgsTagRegisterREAL  (TagManager.ident, TRUE, ADR('dAngleMax'),      SysPar.Sync.dAngleMax);
    PgsTagRegisterREAL  (TagManager.ident, TRUE, ADR('PhaseShift'),     SysPar.Sync.PhaseShift);
    PgsTagEndNode       (TagManager.ident);//sync
    //Bus
    PgsTagStartNode     (TagManager.ident, ADR('exc'));
    PgsTagRegisterREAL  (TagManager.ident, TRUE, ADR('UexcPrim'),     SysPar.Exc.UexcPrim);
    PgsTagRegisterREAL  (TagManager.ident, TRUE, ADR('UexcSec'),      SysPar.Exc.UexcSec);
    PgsTagRegisterREAL  (TagManager.ident, TRUE, ADR('UexcNom'),      SysPar.Exc.UexcNom);
    PgsTagEndNode       (TagManager.ident);//bus
    //Gen
    PgsTagStartNode     (TagManager.ident, ADR('gen'));
    PgsTagRegisterREAL  (TagManager.ident, TRUE, ADR('UmPrim'),     SysPar.Gen.UmPrim);
    PgsTagRegisterREAL  (TagManager.ident, TRUE, ADR('UmSec'),      SysPar.Gen.UmSec);
    PgsTagRegisterREAL  (TagManager.ident, TRUE, ADR('ImPrim'),     SysPar.Gen.ImPrim);
    PgsTagRegisterREAL  (TagManager.ident, TRUE, ADR('ImSec'),      SysPar.Gen.ImSec);
    PgsTagRegisterREAL  (TagManager.ident, TRUE, ADR('UmNom'),      SysPar.Gen.UmNom);
    PgsTagRegisterREAL  (TagManager.ident, TRUE, ADR('SmNom'),      SysPar.Gen.SmNom);
    PgsTagRegisterREAL  (TagManager.ident, TRUE, ADR('FmNom'),      SysPar.Gen.FmNom);
    PgsTagRegisterREAL  (TagManager.ident, TRUE, ADR('UfMin'),      SysPar.Gen.UfMin);
    PgsTagRegisterREAL  (TagManager.ident, TRUE, ADR('UfMax'),      SysPar.Gen.UfMax);
    PgsTagRegisterREAL  (TagManager.ident, TRUE, ADR('UfNom'),      SysPar.Gen.UfNom);
    PgsTagRegisterREAL  (TagManager.ident, TRUE, ADR('IfMin'),      SysPar.Gen.IfMin);
    PgsTagRegisterREAL  (TagManager.ident, TRUE, ADR('IfMax'),      SysPar.Gen.IfMax);
    PgsTagRegisterREAL  (TagManager.ident, TRUE, ADR('IfNom'),      SysPar.Gen.IfNom);
    PgsTagRegisterREAL  (TagManager.ident, TRUE, ADR('RpmNom'),     SysPar.Gen.RpmNom);
    PgsTagRegisterREAL  (TagManager.ident, TRUE, ADR('PPR1'),       SysPar.Gen.PPR1);
    PgsTagRegisterREAL  (TagManager.ident, TRUE, ADR('Pos1_0p'),    SysPar.Gen.Pos1_0p);
    PgsTagRegisterREAL  (TagManager.ident, TRUE, ADR('Pos1_100p'),  SysPar.Gen.Pos1_100p);
    PgsTagRegisterREAL  (TagManager.ident, TRUE, ADR('Pos2_0p'),    SysPar.Gen.Pos2_0p);
    PgsTagRegisterREAL  (TagManager.ident, TRUE, ADR('Pos2_100p'),  SysPar.Gen.Pos2_100p);
    PgsTagRegisterREAL  (TagManager.ident, TRUE, ADR('Pos3_0p'),    SysPar.Gen.Pos3_0p);
    PgsTagRegisterREAL  (TagManager.ident, TRUE, ADR('Pos3_100p'),  SysPar.Gen.Pos3_100p);
    PgsTagRegisterREAL  (TagManager.ident, TRUE, ADR('ClockWise'),  SysPar.Gen.ClockWise);
    PgsTagRegisterREAL  (TagManager.ident, TRUE, ADR('Connection'), SysPar.Gen.Connection);
    PgsTagRegisterREAL  (TagManager.ident, TRUE, ADR('dRpm1Max'),   SysPar.Gen.dRpm1Max);
    PgsTagRegisterREAL  (TagManager.ident, TRUE, ADR('PPR2'),       SysPar.Gen.PPR2);
    PgsTagRegisterREAL  (TagManager.ident, TRUE, ADR('dRpm2Max'),   SysPar.Gen.dRpm2Max);
    PgsTagEndNode       (TagManager.ident);//gen
    //IO
    PgsTagStartNode     (TagManager.ident, ADR('io'));
    PgsTagRegisterREAL  (TagManager.ident, TRUE, ADR('AI1Type'),    SysIOPar.AI1Type);
    PgsTagRegisterREAL  (TagManager.ident, TRUE, ADR('AI2Type'),    SysIOPar.AI2Type);
    PgsTagRegisterREAL  (TagManager.ident, TRUE, ADR('AI3Type'),    SysIOPar.AI3Type);
    PgsTagRegisterREAL  (TagManager.ident, TRUE, ADR('AI4Type'),    SysIOPar.AI4Type);
    PgsTagRegisterREAL  (TagManager.ident, TRUE, ADR('AO1Type'),    SysIOPar.AO1Type);
    PgsTagRegisterREAL  (TagManager.ident, TRUE, ADR('AO2Type'),    SysIOPar.AO2Type);
    PgsTagRegisterREAL  (TagManager.ident, TRUE, ADR('AO3Type'),    SysIOPar.AO3Type);
    PgsTagRegisterREAL  (TagManager.ident, TRUE, ADR('AO4Type'),    SysIOPar.AO4Type);
    PgsTagRegisterREAL  (TagManager.ident, TRUE, ADR('AO1min'),     SysIOPar.AO1min);
    PgsTagRegisterREAL  (TagManager.ident, TRUE, ADR('AO1max'),     SysIOPar.AO1max);
    PgsTagRegisterREAL  (TagManager.ident, TRUE, ADR('AO2min'),     SysIOPar.AO2min);
    PgsTagRegisterREAL  (TagManager.ident, TRUE, ADR('AO2max'),     SysIOPar.AO2max);
    PgsTagRegisterREAL  (TagManager.ident, TRUE, ADR('AO3min'),     SysIOPar.AO3min);
    PgsTagRegisterREAL  (TagManager.ident, TRUE, ADR('AO3max'),     SysIOPar.AO3max);
    PgsTagRegisterREAL  (TagManager.ident, TRUE, ADR('AO4min'),     SysIOPar.AO4min);
    PgsTagRegisterREAL  (TagManager.ident, TRUE, ADR('AO4max'),     SysIOPar.AO4max);
    PgsTagEndNode       (TagManager.ident);//io

    PgsTagEndNode       (TagManager.ident);//system

    SysUpdate.UpdateAll := TRUE;

	//Horimetro
    PgsTagStartNode     (TagManager.ident, ADR('Horimetro'));
    PgsTagRegisterREAL  (TagManager.ident, TRUE, ADR('running_total'),	hour_running.set_total);
    PgsTagRegisterREAL  (TagManager.ident, TRUE, ADR('online_total'),	hour_online.set_total);
	PgsTagEndNode       (TagManager.ident);//Horimetro

	//Energia
    PgsTagStartNode     (TagManager.ident, ADR('Energia'));
    PgsTagRegisterREAL  (TagManager.ident, TRUE, ADR('ativa_pos'),				energia_ativa.set_posEnergy);
    PgsTagRegisterREAL  (TagManager.ident, TRUE, ADR('ativa_neg'),				energia_ativa.set_negEnergy);
    PgsTagRegisterREAL  (TagManager.ident, TRUE, ADR('reativa_pos'),			energia_reativa.set_posEnergy);
    PgsTagRegisterREAL  (TagManager.ident, TRUE, ADR('reativa_neg'),			energia_reativa.set_negEnergy);
	PgsTagEndNode       (TagManager.ident);//Energia

END_PROGRAM
```

### Share.var
```iecst
(*I/O*)
VAR
	A65 : PgsA65;
END_VAR
(*Controls*)
VAR
	avr : PgsAVR := (Parameter:=(CtrlManual:=(CmIf:=(Enable:=FALSE,dRefOn:=0.1,dRefOff:=0.1,PID:=(Kp:=0.004,Ti:=0.05,Td:=0.0,Tf:=1.0,Kwd:=1.2)),CmUf:=(Enable:=FALSE,dRefOn:=0.1,dRefOff:=0.1,PID:=(Kp:=0.002,Ti:=0.05,Td:=0.0,Tf:=1.0,Kwd:=1.2)),CmIm:=(Enable:=FALSE),Ctrl:=PGS_AVR_CM_OFF,EnableOL:=FALSE),CtrlAuto:=(SoftStart:=(RefUm:=1.0,dRefOn:=0.05,dRefOff:=0.0,Offset:=0,RefUm0:=0.3948,FFTmin:=0,FFTmax:=5.0),CaUm0:=(Enable:=FALSE,Ref:=1.0,RefMax:=1.2,RefMin:=0.8,dRefOn:=0.07,dRefOff:=0.07,Kdp:=0.0,PID:=(Kp:=0.003,Ti:=0.1,Td:=0.05,Tf:=1.0,Kwd:=1.2)),CaUm1:=(Enable:=FALSE),CaQm:=(Enable:=FALSE,Ref:=-0.08,RefMax:=0.5,RefMin:=-0.5,dRefOn:=0.01,dRefOff:=0.01,PID:=(Kp:=0.0006,Ti:=1.0,Td:=0.0,Tf:=1.0,Kwd:=1.2),L2max:=1.2,L2min:=0.8,Kdp:=0.1,PIDU:=(Kp:=0.002,Ti:=0.1,Td:=0.05,Tf:=1.0,Kwd:=1.2)),CaPf:=(Enable:=FALSE,Ref:=-0.1,RefMax:=0.3,RefMin:=-0.3,dRefOn:=0.05,dRefOff:=0.05,PID:=(Kp:=0.0006,Ti:=0.8,Td:=0.0,Tf:=1.0,Kwd:=1.2),L2max:=1.2,L2min:=0.8,Kdp:=0.1,PIDU:=(Kp:=0.002,Ti:=0.09,Td:=0.05,Tf:=1.0,Kwd:=1.2))),Limiter:=(Luh:=(Enable:=FALSE,Un:=1.0,Fn:=0.98,Kuh:=1.0,PID:=(Kp:=0.003,Ti:=0.1,Td:=0.05,Tf:=1.0,Kwd:=1.2)),Lifh:=(Enable:=FALSE,SetPoint:=1.1312,Curve:=PGS_AVR_CV_00,Time:=10.0,PID:=(Kp:=0.004,Ti:=0.05,Td:=0.0,Tf:=1.0,Kwd:=1.2)),Lifl:=(Enable:=FALSE,SetPoint:=0.2262,PID:=(Kp:=0.004,Ti:=0.05,Td:=0.0,Tf:=1.0,Kwd:=1.2)),Lifhh:=(Enable:=FALSE,SetPoint:=1.3574,PID:=(Kp:=0.004,Ti:=0.05,Td:=0.0,Tf:=1.0,Kwd:=1.2)),Limh:=(Enable:=FALSE),Lpq:=(Enable:=FALSE))),CtrlOnline:=PGS_AVR_CA_PF);
	gov : PgsGOV := (Parameter:=(CtrlManual:=(CmPos:=(Enable:=FALSE,dRefOn:=0.1,dRefOff:=0.1,RefMax:=1.0,RefMin:=0.0)),CtrlAuto:=(SoftStart:=(Pos0:=0.25,dPos:=0.1,Rpm0:=0.0,Rpm1:=0.2,Rpm2:=0.8,RpmBrake:=0.0,dRpmOn:=0.05,dRpmOff:=0.05,TRpm1:=120,TRpm2:=300),CaRpm0:=(Enable:=FALSE,Ref:=1.0,RefMax:=1.2,RefMin:=0.0,dRefOn:=0.05,dRefOff:=0.05,Kdp:=0.0,PosMax:=0.95,PID:=(Kp:=0.003,Ti:=0.15,Td:=0.0,Tf:=1.0,Kwd:=1.0)),CaRpm1:=(Enable:=FALSE,Ref:=1.025,RefMax:=1.1,RefMin:=0.9,dRefOn:=0.01,dRefOff:=0.01,Kdp:=0.1,PosMax:=0.95,PID:=(Kp:=0.003,Ti:=0.15,Td:=0.0,Tf:=1.0,Kwd:=1.0)),CaHz0:=(Enable:=FALSE,UmOn:=0.5,Ref:=1.0,RefMax:=1.2,RefMin:=0.9,dRefOn:=0.01,dRefOff:=0.1,Kdp:=0.0,PosMax:=0.95,PID:=(Kp:=0.002,Ti:=0.2,Td:=0.5,Tf:=1.0,Kwd:=1.0)),CaHz1:=(Enable:=FALSE,UmOn:=0.5,Ref:=1.025,RefMax:=1.2,RefMin:=0.9,dRefOn:=0.01,dRefOff:=0.01,Kdp:=0.1,PosMax:=0.95,PID:=(Kp:=0.003,Ti:=0.15,Td:=0.0,Tf:=1.0,Kwd:=1.0)),CaPwr:=(Enable:=FALSE,UmOn:=0.5,Ref:=0.02,RefMax:=1.05,RefMin:=0.0,dRefOn:=0.01,dRefOff:=0.01,PID:=(Kp:=0.001,Ti:=0.8,Td:=0.0,Tf:=1.0,Kwd:=1.0),L2max:=1.1,L2min:=0.9,Kdp:=0.1,PosMax:=0.8,PIDHz:=(Kp:=0.002,Ti:=0.2,Td:=0.5,Tf:=1.0,Kwd:=1.0)))),CtrlOnline:=PGS_GOV_CA_PWR);
	pos1 : PgsPOS := (Parameter:=(Enable:=FALSE,Base:=100,RampUp:=(dSp0:=0.1,SetPoint:=0.2,dSp1:=0.3),RampDown:=(dSp0:=0.05,SetPoint:=0.15,dSp1:=0.2),HCC:=(Kup:=1.0,Kdown:=1.0,dbHigh:=0.55,dbLow:=0.45),PID:=(Kp:=0.05,Ti:=5.0,Td:=0.0,Tf:=1.0,Kwd:=1.0,Update:=TRUE)));
	pos2 : PgsPOS := (Parameter:=(Enable:=FALSE,Base:=100,RampUp:=(dSp0:=0.1,SetPoint:=0.2,dSp1:=0.3),RampDown:=(dSp0:=0.05,SetPoint:=0.15,dSp1:=0.2),HCC:=(Kup:=1.0,Kdown:=1.0,dbHigh:=0.55,dbLow:=0.45),PID:=(Kp:=0.05,Ti:=5.0,Td:=0.0,Tf:=1.0,Kwd:=1.0,Update:=TRUE)));
	pos3 : PgsPOS := (Parameter:=(Enable:=FALSE,Base:=100,RampUp:=(dSp0:=0.1,SetPoint:=0.2,dSp1:=0.3),RampDown:=(dSp0:=0.05,SetPoint:=0.15,dSp1:=0.2),HCC:=(Kup:=1.0,Kdown:=1.0,dbHigh:=0.55,dbLow:=0.45),PID:=(Kp:=0.05,Ti:=5.0,Td:=0.0,Tf:=1.0,Kwd:=1.0,Update:=TRUE)));
	curve1 : PgsCurve := (Curve:=(in:=[0.0,0.2,0.3,0.4,0.5,0.6,0.7,0.8,0.9,1.0],out:=[0.0,0.2,0.3,0.4,0.5,0.6,0.7,0.8,0.9,1.0]));
	curve2 : PgsCurve := (Curve:=(in:=[0.0,0.2,0.3,0.4,0.5,0.6,0.7,0.8,0.9,1.0],out:=[0.0,0.2,0.3,0.4,0.5,0.6,0.7,0.8,0.9,1.0]));
	curve3 : PgsCurve := (Curve:=(in:=[0.0,0.2,0.3,0.4,0.5,0.6,0.7,0.8,0.9,1.0],out:=[0.0,0.2,0.3,0.4,0.5,0.6,0.7,0.8,0.9,1.0]));
END_VAR
(*Protection*)
VAR
	phaseFault : PgsProtPhaseFault;
END_VAR
(*Meter*)
VAR
	meter : PgsMeter := (Base:=(Sm:=1000,Um:=380,Fm:=60,Rot:=2000,Uf:=80,If:=10));
	filter_uf : LCRMovAvgFlt;
	pos1_input : REAL;
	pos2_input : REAL;
	pos3_input : REAL;
	uf_input : REAL;
	if_input : REAL;
END_VAR
(*Hour Meter*)
VAR
	hour_running : PgsHorimetro;
	hour_online : PgsHorimetro;
END_VAR
(*Energy Meter*)
VAR
	energia_ativa : PgsEnergia;
	energia_reativa : PgsEnergia;
	energy_active : PgsEnergy;
	energy_reactive : PgsEnergy;
END_VAR
```

### Share.typ
```iecst
TYPE
	PgsA65 : 	STRUCT
		di : PgsA65DI;
		do : PgsA65DO;
		ai : PgsA65AI;
		ao : PgsA65AO;
	END_STRUCT;
	PgsA65DI : 	STRUCT
		remote : BOOL;
		reset : BOOL;
		gov_enable : BOOL;
		gov_ctrl_pwr_enable : BOOL;
		gov_trip : BOOL;
		gov_unload : BOOL;
		gov_up : BOOL;
		gov_down : BOOL;
		avr_enable : BOOL;
		avr_ctrl_qm_enable : BOOL;
		avr_ctrl_pf_enable : BOOL;
		avr_trip : BOOL;
		avr_unload : BOOL;
		avr_ref_up : BOOL;
		avr_ref_down : BOOL;
		sync_enable : BOOL;
		dead_bus_enable : BOOL;
		enable_pos1 : BOOL;
		enable_pos2 : BOOL;
		enable_pos3 : BOOL;
	END_STRUCT;
	PgsA65DO : 	STRUCT
		gov_on : BOOL;
		gov_unload : BOOL;
		gov_over_rotation : BOOL;
		rotation_zero : BOOL;
		rotation_nominal : BOOL;
		rotation_brake : BOOL;
		power_zero : BOOL;
		rpm_fault : BOOL;
		avr_on : BOOL;
		avr_force_crowbar : BOOL;
		avr_limiter_on : BOOL;
		field_flash_on : BOOL;
		voltage_nominal : BOOL;
		sync_enabled : BOOL;
		dead_bus_enabled : BOOL;
		watchdog : BOOL;
	END_STRUCT;
	PgsA65AI : 	STRUCT
		if : INT;
		uf : INT;
		pos1 : INT;
		pos2 : INT;
		pos3 : INT;
	END_STRUCT;
	PgsA65AO : 	STRUCT
		pwr : INT;
		pos1 : INT;
		pos2 : INT;
		pos3 : INT;
	END_STRUCT;
END_TYPE
```

### Program Logical/Kontrol/Control/Control (IEC)

#### Cyclic.st - Cyclic code
```iecst
PROGRAM _CYCLIC

    IF NOT PgsTagValid(TagManager.ident) THEN
        RETURN;
    END_IF

	cm0985Meter();

    phaseFault(
        Enable  := TRUE,
        Ph1     := cm0985Meter.Ug1,
        Ph2     := cm0985Meter.Ug2,
        Ph3     := cm0985Meter.Ug3
    );

(*******************************************************
****************** Circuit Breaker  ********************
*******************************************************)
    avr.DigInputs.Online := CB52.st.closed;
    gov.DigInputs.Online := CB52.st.closed;

(******************************************************)
    //Reset
    IF A65.di.reset THEN
        //A65.di.reset        := FALSE;
        avr.DigInputs.Reset := TRUE;
		gov.DigInputs.Reset := TRUE;
		//Reset to Auto Mode
//		gov.DigInputs.Auto  := TRUE;
//		avr.DigInputs.Auto  := TRUE;
    END_IF;

    IF NOT A65.di.remote THEN
        //GOV
        gov.DigInputs.Start     := A65.di.gov_enable;
        gov.DigInputs.Stop      := NOT A65.di.gov_enable;
        gov.DigInputs.Unload    := A65.di.gov_unload;
		gov.DigInputs.RefUp		:= A65.di.gov_up;
		gov.DigInputs.RefDown	:= A65.di.gov_down;
        IF A65.di.gov_ctrl_pwr_enable THEN
            gov.CtrlOnline  := PGS_GOV_CA_PWR;
        ELSE
            gov.CtrlOnline  := PGS_GOV_CA_HZ_1;
        END_IF;

        //AVR
		A65.di.avr_unload		:= A65.di.gov_unload;
        avr.DigInputs.Start     := A65.di.avr_enable;
        avr.DigInputs.Stop      := NOT A65.di.avr_enable;
        avr.DigInputs.Unload    := A65.di.avr_unload;
		avr.DigInputs.RefUp		:= A65.di.avr_ref_up;
		avr.DigInputs.RefDown	:= A65.di.avr_ref_down;

        IF A65.di.avr_ctrl_qm_enable    THEN
            avr.CtrlOnline  := PGS_AVR_CA_QM;
        ELSIF  A65.di.avr_ctrl_pf_enable THEN
            avr.CtrlOnline  := PGS_AVR_CA_PF;
        ELSE
            avr.CtrlOnline  := PGS_AVR_CA_UM_1;
        END_IF;
    END_IF;

    (******************************************************)

	//TRIP
	IF A65.di.avr_trip OR NOT Protection.do.trip_86e THEN
        avr.DigInputs.Stop := TRUE;
    END_IF;
    IF A65.di.gov_trip OR NOT Protection.do.trip_86h THEN
        gov.DigInputs.Stop := TRUE;
    END_IF;

	//Meters

    //Icc ==> fix 4-20mA
    scale_if.x1 := 4.0;
    scale_if.x2 := 20.0;
    if_input	:= IfAvg * 16.0 / 32767.0 + 4.0;

    scale_if(
        x   := if_input,
        y1  := SysPar.Gen.IfMin,
        y2  := SysPar.Gen.IfMax
    );
	meter.In.If := scale_if.y;

	//Vcc ==> fix 4-20mA
    scale_uf.x1 := 4.0;
    scale_uf.x2 := 20.0;
	uf_input	:= UfAvg * 16.0 / 32767.0 + 4.0;
    scale_uf(
        x   := uf_input,
        y1  := SysPar.Gen.UfMin,
        y2  := SysPar.Gen.UfMax
    );
	meter.In.Uf := scale_uf.y;

	filter_uf( x := meter.In.Uf );
    //Ub
    IF cm0985Main.Enable3phase THEN
        meter.In.Ub := (cm0985Meter.Un12 + cm0985Meter.Un23 + cm0985Meter.Un31) / 3;
    ELSE
        meter.In.Ub := cm0985Meter.Un12;
    END_IF;
	//Um
	IF NOT phaseFault.Fault1 AND NOT phaseFault.Fault2 AND NOT phaseFault.Fault3 THEN
        meter.In.Um 	:=  cm0985Meter.Ug;
    ELSIF phaseFault.Fault1 AND NOT phaseFault.Fault2 AND NOT phaseFault.Fault3 THEN
        meter.In.Um 	:=  cm0985Meter.Ug23;
    ELSIF NOT phaseFault.Fault1 AND phaseFault.Fault2 AND NOT phaseFault.Fault3 THEN
        meter.In.Um 	:=  cm0985Meter.Ug31;
    ELSIF NOT phaseFault.Fault1 AND NOT phaseFault.Fault2 AND phaseFault.Fault3 THEN
        meter.In.Um 	:=  cm0985Meter.Ug12;
    ELSE
        meter.In.Um     :=  phaseFault.Phm * SQRT(3);
    END_IF

	meter.In.Im		:= cm0985Meter.Ig;
	IF meter.In.Um < 5 THEN
		meter.In.Fm		:= 0.0;
		meter.In.PF		:= 1.0;
	ELSE
		meter.In.Fm		:= cm0985Meter.Fg;
		meter.In.PF		:= cm0985Meter.PFg;
	END_IF;
	meter.In.Pm		:= cm0985Meter.Pg;
	meter.In.Qm		:= cm0985Meter.Qg;
	meter.In.Sm		:= cm0985Meter.Sg;

    rpm1(ppr := REAL_TO_INT(SysPar.Gen.PPR1));
    filter_rpm1.IN := rpm1.Output;
	filter_rpm1();

    rpm2(ppr := REAL_TO_INT(SysPar.Gen.PPR2));
    IF SysPar.Gen.PPR2 <> 0 THEN
		filter_rpm2.IN := rpm2.Output;
	ELSE
		filter_rpm2.IN := 0.0;
	END_IF;
    filter_rpm2();

	IF filter_rpm1.OUT > filter_rpm2.OUT THEN
	    meter.In.Rot := filter_rpm1.OUT;
    ELSE
	    meter.In.Rot := filter_rpm2.OUT;
    END_IF;

	IF SysPar.Gen.PPR2 <> 0 THEN
		A65.do.rpm_fault := ( ABS(filter_rpm1.OUT - filter_rpm2.OUT) / meter.Base.Rot ) > 0.05;
	ELSE
		A65.do.rpm_fault := FALSE;
	END_IF;
	meter       ();

	//Position
    //pos1 - ==> fix 4-20mA
	pos1_input	    := INT_TO_REAL(A65.ai.pos1) * 16.0 / 32767.0 + 4.0;
	filter_pos1(IN:=pos1_input);
    scale_pos1(
        x   := filter_pos1.OUT,
		x1  := SysPar.Gen.Pos1_0p,
        x2  := SysPar.Gen.Pos1_100p
    );
	pos1.PosIn	:= scale_pos1.y;

    pos2_input	    := INT_TO_REAL(A65.ai.pos2) * 16.0 / 32767.0 + 4.0;
    scale_pos2(
        x   := pos2_input,
		x1  := SysPar.Gen.Pos2_0p,
		x2  := SysPar.Gen.Pos2_100p
	);
	pos2.PosIn	:= scale_pos2.y;

    pos3_input	    := INT_TO_REAL(A65.ai.pos3) * 16.0 / 32767.0 + 4.0;
    scale_pos3(
        x   := pos3_input,
		x1  := SysPar.Gen.Pos3_0p,
		x2  := SysPar.Gen.Pos3_100p
	);
    pos3.PosIn := scale_pos3.y;

	//Syncronizer
    IF A65.di.remote THEN
        cm0985IO.do.SyncSlip    := SysUpdate.EnableSync;
        cm0985IO.do.SyncDeadBus := SysUpdate.EnableDeadBus AND NOT SysUpdate.EnableSync;
    ELSE
        cm0985IO.do.SyncSlip    := A65.di.sync_enable AND NOT CB52.st.closed;
        cm0985IO.do.SyncDeadBus := A65.di.dead_bus_enable AND NOT CB52.st.closed AND NOT A65.di.sync_enable;
    END_IF;
	A65.do.sync_enabled     := cm0985IO.do.SyncSlip OR cm0985IO.do.SyncDeadBus;
    IF cm0985IO.do.SyncSlip THEN
		IF cm0985Meter.dAngle > 15 AND cm0985Meter.dAngle < 345 THEN
			gov.SetPoints.fastSetHz := (cm0985Meter.Fs1 / meter.Base.Fm) * 1.001;
		ELSE
			gov.SetPoints.fastSetHz := cm0985Meter.Fs1 / meter.Base.Fm;
		END_IF;
		avr.SetPoints.fastSetUm := meter.Out.Ub;
	END_IF;

//=======================================================================
//=====	Para maior estabilidade do controle de potência	=================
//=======================================================================
	// Filtro da leitura da potência para estabilizar o sinal
	IF meter.Out.Pm <> 0 THEN
		filter_pwr(IN:=meter.Out.Pm);
	ELSE
		filter_pwr(IN:=0.0001);
	END_IF;
	// Verifica se a diferença em módulo da potência é menor que 2%
	IF  ABS(filter_pwr.OUT - gov.SetPoints.fastSetPwr) < 0.005
		// Verifica se a diferença em módulo do controle é menor que 5%
	AND ABS(1 - gov.SetPoints.fastSetHz) < 0.03	THEN
		// Se a deadband do PID for diferente, aplica deadband
		IF gov.Parameter.CtrlAuto.CaPwr.PID.db <> 0.03 THEN
			gov.Parameter.CtrlAuto.CaPwr.PID.Update		:= TRUE;
			gov.Parameter.CtrlAuto.CaPwr.PIDHz.Update	:= TRUE;
		END_IF;
		gov.Parameter.CtrlAuto.CaPwr.PID.db		:= 0.03;
		gov.Parameter.CtrlAuto.CaPwr.PIDHz.db	:= 0.03;
	ELSE
		// Se a deadband do PID for diferente, desaplica deadband
		IF gov.Parameter.CtrlAuto.CaPwr.PID.db <> 0.00 THEN
			gov.Parameter.CtrlAuto.CaPwr.PID.Update	:= TRUE;
			gov.Parameter.CtrlAuto.CaPwr.PIDHz.Update	:= TRUE;
		END_IF;
		gov.Parameter.CtrlAuto.CaPwr.PID.db		:= 0.00;
		gov.Parameter.CtrlAuto.CaPwr.PIDHz.db	:= 0.01;
	END_IF;

	pwr_tp(IN:= CB52.st.closed, PT:=T#2s);
	IF pwr_tp.Q THEN
		gov.SetPoints.fastSetPwr := 0.1;
	END_IF;
	pwr_ton(IN:= CB52.st.closed AND NOT pwr_mem, PT:= T#5s);
	IF pwr_ton.Q THEN
		pwr_mem := TRUE;
		gov.SetPoints.SetPwr := gov.Parameter.CtrlAuto.CaPwr.Ref;
	END_IF;
	IF NOT CB52.st.closed THEN
		pwr_mem := FALSE;
	END_IF;
//=======================================================================
//=======================================================================

	//GOV
	gov     ();

	//POS1
    curve1	( In := gov.Out);
    pos1	( In := curve1.Out, Enable := (gov.DigOutputs.Status.Enable	AND NOT A65.di.gov_trip)
									OR  pos1.Mode > PGS_POS_MD_AUTO
									OR	A65.di.enable_pos1 );
    //Gov Out1
    IF A65.di.gov_trip THEN
		scale_gov_o1.x := (pos1.Parameter.HCC.dbHigh + pos1.Parameter.HCC.dbLow) / 2.0;
    ELSE
        scale_gov_o1.x := pos1.Out;
    END_IF;
	scale_gov_o1(
		x1 := 0.0,
		x2 := 1.0,
		y1 := 0,
		y2 := 32767.0);
    A65.ao.pos1 := REAL_TO_INT(scale_gov_o1.y);

    //POS2
    curve2	( In := gov.Out );
    pos2	( In := curve2.Out, Enable := (gov.DigOutputs.Status.Enable AND NOT A65.di.gov_trip)
									OR  pos2.Mode <> PGS_POS_MD_AUTO
									OR	A65.di.enable_pos2 );

    //Gov Out2
    IF A65.di.gov_trip THEN
		scale_gov_o2.x := (pos2.Parameter.HCC.dbHigh + pos2.Parameter.HCC.dbLow) / 2.0;
    ELSE
        scale_gov_o2.x := pos2.Out;
    END_IF;
	scale_gov_o2(
		x1 := 0.0,
		x2 := 1.0,
		y1 := 0,
		y2 := 32767.0);
    A65.ao.pos2 := REAL_TO_INT(scale_gov_o2.y);

    //POS3
    curve3	( In := gov.Out );
    pos3	( In := curve3.Out, Enable := (gov.DigOutputs.Status.Enable AND NOT A65.di.gov_trip)
									OR  pos3.Mode <> PGS_POS_MD_AUTO
									OR	A65.di.enable_pos3 );
    //Gov Out3
    IF A65.di.gov_trip THEN
		scale_gov_o3.x := (pos3.Parameter.HCC.dbHigh + pos3.Parameter.HCC.dbLow) / 2.0;
    ELSE
        scale_gov_o3.x := pos3.Out;
    END_IF;
	scale_gov_o3(
		x1 := 0.0,
		x2 := 1.0,
		y1 := 0,
		y2 := 32767.0);
    A65.ao.pos3 := REAL_TO_INT(scale_gov_o3.y);

    //Gov Pos feedback
    gov.PosIn   := pos1.PosOut;

    //Digital Outputs
    A65.do.gov_on               := gov.DigOutputs.Status.Enable;
    A65.do.rotation_zero        := meter.Out.Rot <= 0.01; //gov.DigOutputs.Status.Stopped;
    A65.do.rotation_nominal     := gov.DigOutputs.Status.RotationOk;
    A65.do.rotation_brake       := gov.DigOutputs.Status.RotationBrake;
    A65.do.gov_unload           := gov.DigOutputs.Status.Unloaded;
    A65.do.gov_over_rotation    := gov.DigOutputs.Trip.OverRotation;
    A65.do.power_zero           := meter.Out.Pm < gov.Parameter.CtrlAuto.CaPwr.RefOpen;

	//AVR
    avr			();
    //Avr Out1
	scale_avr_o1(
		x  := avr.Out,
		x1 := 0.0,
		x2 := 1.0,
		y1 := 0,
		y2 := 32767.0);
    A65.ao.pwr := REAL_TO_INT(scale_avr_o1.y);

    //Digital Outputs
    A65.do.avr_on               := avr.DigOutputs.Status.Enable;
    A65.do.field_flash_on	    := avr.DigOutputs.Status.FieldFlashOn;
	A65.do.voltage_nominal      := avr.DigOutputs.Status.VoltageOK;
    A65.do.avr_force_crowbar    := A65.di.avr_trip OR NOT avr.DigOutputs.Status.Enable;
    A65.do.avr_limiter_on       := avr.DigOutputs.Alarm.LimiterMin OR avr.DigOutputs.Alarm.LimiterMax;

//***************************************************
//****************** Hour Meter  ********************
//***************************************************
	hour_running	( enable := meter.Out.Rot > 0 ); // Maybe put frequency too?
	hour_online		( enable := gov.DigInputs.Online OR avr.DigInputs.Online );

//***************************************************
//**************** Energy Meter  ********************
//***************************************************
	energy_active	(
		enable	:= TRUE,
		power	:= meter.In.Pm
	);
	energy_reactive	(
		enable	:= TRUE,
		power	:= meter.In.Qm
	);

END_PROGRAM
```

#### Init.st - Init code
```iecst
PROGRAM _INIT

    TagManager(enable:=TRUE);

//    EvtGroup.enable     := TRUE;
//    EvtGroup.group      := ADR('Control');
//    EvtGroup.pData      := ADR(EvtMemory);
//    EvtGroup.dataSize   := SIZEOF(EvtMemory);

    //Meter Base
	meter();

	//Curve1
	curve1();
	link_curve1.CurveIdent	:= curve1.Ident;
    PgsTagRegisterCurve(TagManager.ident, ADR('curve1'), curve1);

	//Curve2
	curve2();
	link_curve2.CurveIdent	:= curve2.Ident;
    PgsTagRegisterCurve(TagManager.ident, ADR('curve2'), curve2);

	//Curve3
	curve3();
	link_curve3.CurveIdent	:= curve3.Ident;
    PgsTagRegisterCurve(TagManager.ident, ADR('curve3'), curve3);

	//Pos3:
	pos3.Mode				:= PGS_POS_MD_AUTO;
	pos3.PosIdent			:= 0;
	pos3();
	link_pos3.PosIdent		:= pos3.Ident;
    PgsTagRegisterPOS(TagManager.ident, ADR('pos3'), pos3);

	//POS3
	scale_pos3.y1			:= 0.0;
	scale_pos3.y2			:= 100.0;

	//Po2:
	pos2.Mode				:= PGS_POS_MD_AUTO;
	pos2.PosIdent			:= pos3.Ident;
	pos2();
	link_pos2.PosIdent		:= pos2.Ident;
    PgsTagRegisterPOS(TagManager.ident, ADR('pos2'), pos2);

	//POS2
	scale_pos2.y1			:= 0.0;
	scale_pos2.y2			:= 100.0;

	//Pos1:
	pos1.Mode				:= PGS_POS_MD_AUTO;
	pos1.PosIdent			:= pos2.Ident;
	pos1();
	link_pos1.PosIdent		:= pos1.Ident;
    PgsTagRegisterPOS(TagManager.ident, ADR('pos1'), pos1);

	//POS1
	scale_pos1.y1			:= 0.0;
    scale_pos1.y2			:= 100.0;

	//GOV
	gov.DigInputs.Auto		:= TRUE;
	gov.MeterIdent          := meter.Ident;
	gov.PosIdent			:= pos1.Ident;
    gov.CtrlOnline          := PGS_GOV_CA_PWR;
	gov();
	link_gov.GovIdent	    := gov.Ident;
    PgsTagRegisterGOV(TagManager.ident, ADR('gov'), gov);

    //RPM
	filter_rpm1.CTE 	    := 32;
	filter_rpm2.CTE 	    := 32;

	//AVR
	avr.DigInputs.Auto		:=	TRUE;
    avr.MeterIdent          := meter.Ident;
    avr.CtrlOnline          := PGS_AVR_CA_QM;
    avr();
	link_avr.AvrIdent       := avr.Ident;
    PgsTagRegisterAVR(TagManager.ident, ADR('avr'), avr);

	//field
	filter_uf.enable	    := TRUE;
	filter_uf.base 	        := 32;
	filter_uf();

	A65.di.gov_ctrl_pwr_enable	:= TRUE;
	A65.di.avr_ctrl_qm_enable	:= TRUE;

	//Meter Register
    PgsTagStartNode     (TagManager.ident, ADR('meter'));
    PgsTagRegisterREAL  (TagManager.ident, FALSE, ADR('Um'),        meter.In.Um);
    PgsTagRegisterREAL  (TagManager.ident, FALSE, ADR('Im'),        meter.In.Im);
    PgsTagRegisterREAL  (TagManager.ident, FALSE, ADR('Pm'),        meter.In.Pm);
    PgsTagRegisterREAL  (TagManager.ident, FALSE, ADR('Qm'),        meter.In.Qm);
    PgsTagRegisterREAL  (TagManager.ident, FALSE, ADR('Sm'),        meter.In.Sm);
    PgsTagRegisterREAL  (TagManager.ident, FALSE, ADR('PF'),        meter.In.PF);
    PgsTagRegisterREAL  (TagManager.ident, FALSE, ADR('Fm'),        meter.In.Fm);
    PgsTagRegisterREAL  (TagManager.ident, FALSE, ADR('Uf'),        meter.In.Uf);
    PgsTagRegisterREAL  (TagManager.ident, FALSE, ADR('If'),        meter.In.If);
    PgsTagRegisterREAL  (TagManager.ident, FALSE, ADR('Rot'),       meter.In.Rot);
    PgsTagRegisterREAL  (TagManager.ident, FALSE, ADR('Pos1'),      pos1.PosIn);
    PgsTagRegisterREAL  (TagManager.ident, FALSE, ADR('Pos2'),      pos2.PosIn);
    PgsTagRegisterREAL  (TagManager.ident, FALSE, ADR('Pos3'),      pos3.PosIn);
    PgsTagEndNode       (TagManager.ident);//meter

END_PROGRAM
```

#### Variables.var - Local variables
```iecst
(*Pwr*)
VAR
	pwr_tp : TP;
	pwr_ton : TON;
	pwr_mem : BOOL;
END_VAR
(*RPM Inputs*)
VAR
	rpm1 : PgsRPM;
	rpm2 : PgsRPM;
	filter_rpm1 : PgsFiltro;
	filter_rpm2 : PgsFiltro;
END_VAR
(*Analog Inputs*)
VAR
	scale_if : LCRScal;
	scale_uf : LCRScal;
	scale_pos1 : LCRScal;
	scale_pos2 : LCRScal;
	scale_pos3 : LCRScal;
	filter_pos1 : PgsFiltro := (CTE:=20);
	filter_pwr : PgsFiltro := (CTE:=100);
END_VAR
(*Analog Outputs*)
VAR
	scale_avr_o1 : LCRScal;
	scale_gov_o1 : LCRScal;
	scale_gov_o2 : LCRScal;
	scale_gov_o3 : LCRScal;
END_VAR
```

### Share.var
```iecst
VAR
	CB52 : PgsCb52;
END_VAR
```

### Program Logical/Kontrol/CB52/cb52 (IEC)

#### Cyclic.st
```iecst
PROGRAM _CYCLIC

    CB52.st.closed  := CB52.di.closed;
    CB52.st.opened  := NOT CB52.di.closed;

END_PROGRAM
```

### Share.typ
```iecst
TYPE
	PgsProtType : 	STRUCT
		di : PgsProtDiType;
		do : PgsProtDoType;
		ai : PgsProtAiType;
	END_STRUCT;
	PgsProtDiType : 	STRUCT
		reset : BOOL;
		crowbar_ok : BOOL;
		pwr_temp_ok : BOOL;
		relay_86E_ok : BOOL;
	END_STRUCT;
	PgsProtDoType : 	STRUCT
		trip_86e : BOOL;
		trip_86h : BOOL;
		trip_50bf : BOOL;
	END_STRUCT;
	PgsProtAiType : 	STRUCT
		ExcTemp : INT;
	END_STRUCT;
	PgsProtParType : 	STRUCT
		P59P_L1 : REAL; (*Phase V in p.u.*)
		T59P_L1 : REAL; (*second*)
		P59PP_L1 : REAL; (*Phase-Phase V in p.u.*)
		T59PP_L1 : REAL; (*second*)
		P59V1_L1 : REAL; (*Phase V in p.u.*)
		T59V1_L1 : REAL; (*second*)
		P59Q_L1 : REAL; (*Phase V in p.u.*)
		T59Q_L1 : REAL; (*second*)
		P59G_L1 : REAL; (*Phase V in p.u.*)
		T59G_L1 : REAL; (*second*)
		P59P_L2 : REAL; (*Phase V in p.u.*)
		T59P_L2 : REAL; (*second*)
		P59PP_L2 : REAL; (*Phase-Phase V in p.u.*)
		T59PP_L2 : REAL; (*second*)
		P59V1_L2 : REAL; (*Phase V in p.u.*)
		T59V1_L2 : REAL; (*second*)
		P59Q_L2 : REAL; (*Phase V in p.u.*)
		T59Q_L2 : REAL; (*second*)
		P59G_L2 : REAL; (*Phase V in p.u.*)
		T59G_L2 : REAL; (*second*)
		P27P_L1 : REAL; (*Phase V in p.u.*)
		T27P_L1 : REAL; (*second*)
		P27PP_L1 : REAL; (*Phase-Phase V in p.u.*)
		T27PP_L1 : REAL; (*second*)
		P27V1_L1 : REAL; (*Phase V in p.u.*)
		T27V1_L1 : REAL; (*second*)
		P27P_L2 : REAL; (*Phase V in p.u.*)
		T27P_L2 : REAL; (*second*)
		P27PP_L2 : REAL; (*Phase-Phase V in p.u.*)
		T27PP_L2 : REAL; (*second*)
		P27V1_L2 : REAL; (*Phase V in p.u.*)
		T27V1_L2 : REAL; (*second*)
		P81O_L1 : REAL;
		T81O_L1 : REAL;
		P81O_L2 : REAL;
		T81O_L2 : REAL;
		P81U_L1 : REAL;
		T81U_L1 : REAL;
		P81U_L2 : REAL;
		T81U_L2 : REAL;
		P32OP_L1 : REAL;
		T32OP_L1 : REAL;
		P32UP_L1 : REAL;
		T32UP_L1 : REAL;
		P32OQ_L1 : REAL;
		T32OQ_L1 : REAL;
		P32UQ_L1 : REAL;
		T32UQ_L1 : REAL;
		P50P_L1 : REAL;
		T50P_L1 : REAL;
		P50Q_L1 : REAL;
		T50Q_L1 : REAL;
		P50G_L1 : REAL;
		T50G_L1 : REAL;
		P50P_L2 : REAL;
		T50P_L2 : REAL;
		P50Q_L2 : REAL;
		T50Q_L2 : REAL;
		P50G_L2 : REAL;
		T50G_L2 : REAL;
		P51V_L1 : REAL;
		T51V_L1 : REAL;
		C51V_L1 : REAL;
		P51P_L1 : REAL;
		T51P_L1 : REAL;
		C51P_L1 : REAL;
		P51Q_L1 : REAL;
		T51Q_L1 : REAL;
		C51Q_L1 : REAL;
		P51G_L1 : REAL;
		T51G_L1 : REAL;
		C51G_L1 : REAL;
		P24_L1 : REAL;
		T24_L1 : REAL;
		D40_L1 : REAL;
		O40_L1 : REAL;
		T40_L1 : REAL;
		D40_L2 : REAL;
		O40_L2 : REAL;
		T40_L2 : REAL;
		T50BF : REAL;
	END_STRUCT;
	PgsProtFlagType : 	STRUCT
		KeyInvalid : BOOL;
		WatchDog : BOOL;
		GenPhAFault : BOOL;
		GenPhBFault : BOOL;
		GenPhCFault : BOOL;
		ExcPhAFault : BOOL;
		ExcPhBFault : BOOL;
		ExcPhCFault : BOOL;
		ExcCrowBar : BOOL;
		ExcOverTemp : BOOL;
		UgPhSeqFault : BOOL;
		IgPhSeqFault : BOOL;
		Us1PhSeqFault : BOOL;
		PwrSrcCpuIOFault : BOOL;
		PwrSrcM1IOFault : BOOL;
		M1Fault : BOOL;
		M2Fault : BOOL;
		M3Fault : BOOL;
		T86E : BOOL;
		T86H : BOOL;
		P59A_L1 : BOOL;
		T59A_L1 : BOOL;
		L59A_L1 : BOOL;
		P59B_L1 : BOOL;
		T59B_L1 : BOOL;
		L59B_L1 : BOOL;
		P59C_L1 : BOOL;
		T59C_L1 : BOOL;
		L59C_L1 : BOOL;
		P59AB_L1 : BOOL;
		T59AB_L1 : BOOL;
		L59AB_L1 : BOOL;
		P59BC_L1 : BOOL;
		T59BC_L1 : BOOL;
		L59BC_L1 : BOOL;
		P59CA_L1 : BOOL;
		T59CA_L1 : BOOL;
		L59CA_L1 : BOOL;
		P59V1_L1 : BOOL;
		T59V1_L1 : BOOL;
		L59V1_L1 : BOOL;
		P59Q_L1 : BOOL;
		T59Q_L1 : BOOL;
		L59Q_L1 : BOOL;
		P59G_L1 : BOOL;
		T59G_L1 : BOOL;
		L59G_L1 : BOOL;
		P59A_L2 : BOOL;
		T59A_L2 : BOOL;
		L59A_L2 : BOOL;
		P59B_L2 : BOOL;
		T59B_L2 : BOOL;
		L59B_L2 : BOOL;
		P59C_L2 : BOOL;
		T59C_L2 : BOOL;
		L59C_L2 : BOOL;
		P59AB_L2 : BOOL;
		T59AB_L2 : BOOL;
		L59AB_L2 : BOOL;
		P59BC_L2 : BOOL;
		T59BC_L2 : BOOL;
		L59BC_L2 : BOOL;
		P59CA_L2 : BOOL;
		T59CA_L2 : BOOL;
		L59CA_L2 : BOOL;
		P59V1_L2 : BOOL;
		T59V1_L2 : BOOL;
		L59V1_L2 : BOOL;
		P59Q_L2 : BOOL;
		T59Q_L2 : BOOL;
		L59Q_L2 : BOOL;
		P59G_L2 : BOOL;
		T59G_L2 : BOOL;
		L59G_L2 : BOOL;
		P27A_L1 : BOOL;
		T27A_L1 : BOOL;
		L27A_L1 : BOOL;
		P27B_L1 : BOOL;
		T27B_L1 : BOOL;
		L27B_L1 : BOOL;
		P27C_L1 : BOOL;
		T27C_L1 : BOOL;
		L27C_L1 : BOOL;
		P27AB_L1 : BOOL;
		T27AB_L1 : BOOL;
		L27AB_L1 : BOOL;
		P27BC_L1 : BOOL;
		T27BC_L1 : BOOL;
		L27BC_L1 : BOOL;
		P27CA_L1 : BOOL;
		T27CA_L1 : BOOL;
		L27CA_L1 : BOOL;
		P27V1_L1 : BOOL;
		T27V1_L1 : BOOL;
		L27V1_L1 : BOOL;
		P27A_L2 : BOOL;
		T27A_L2 : BOOL;
		L27A_L2 : BOOL;
		P27B_L2 : BOOL;
		T27B_L2 : BOOL;
		L27B_L2 : BOOL;
		P27C_L2 : BOOL;
		T27C_L2 : BOOL;
		L27C_L2 : BOOL;
		P27AB_L2 : BOOL;
		T27AB_L2 : BOOL;
		L27AB_L2 : BOOL;
		P27BC_L2 : BOOL;
		T27BC_L2 : BOOL;
		L27BC_L2 : BOOL;
		P27CA_L2 : BOOL;
		T27CA_L2 : BOOL;
		L27CA_L2 : BOOL;
		P27V1_L2 : BOOL;
		T27V1_L2 : BOOL;
		L27V1_L2 : BOOL;
		P81O_L1 : BOOL;
		T81O_L1 : BOOL;
		L81O_L1 : BOOL;
		P81O_L2 : BOOL;
		T81O_L2 : BOOL;
		L81O_L2 : BOOL;
		P81U_L1 : BOOL;
		T81U_L1 : BOOL;
		L81U_L1 : BOOL;
		P81U_L2 : BOOL;
		T81U_L2 : BOOL;
		L81U_L2 : BOOL;
		P32OP_L1 : BOOL;
		T32OP_L1 : BOOL;
		L32OP_L1 : BOOL;
		P32UP_L1 : BOOL;
		T32UP_L1 : BOOL;
		L32UP_L1 : BOOL;
		P32OQ_L1 : BOOL;
		T32OQ_L1 : BOOL;
		L32OQ_L1 : BOOL;
		P32UQ_L1 : BOOL;
		T32UQ_L1 : BOOL;
		L32UQ_L1 : BOOL;
		P50PA_L1 : BOOL;
		T50PA_L1 : BOOL;
		L50PA_L1 : BOOL;
		P50PB_L1 : BOOL;
		T50PB_L1 : BOOL;
		L50PB_L1 : BOOL;
		P50PC_L1 : BOOL;
		T50PC_L1 : BOOL;
		L50PC_L1 : BOOL;
		P50Q_L1 : BOOL;
		T50Q_L1 : BOOL;
		L50Q_L1 : BOOL;
		P50G_L1 : BOOL;
		T50G_L1 : BOOL;
		L50G_L1 : BOOL;
		P50PA_L2 : BOOL;
		T50PA_L2 : BOOL;
		L50PA_L2 : BOOL;
		P50PB_L2 : BOOL;
		T50PB_L2 : BOOL;
		L50PB_L2 : BOOL;
		P50PC_L2 : BOOL;
		T50PC_L2 : BOOL;
		L50PC_L2 : BOOL;
		P50Q_L2 : BOOL;
		T50Q_L2 : BOOL;
		L50Q_L2 : BOOL;
		P50G_L2 : BOOL;
		T50G_L2 : BOOL;
		L50G_L2 : BOOL;
		P51VA_L1 : BOOL;
		T51VA_L1 : BOOL;
		R51VA_L1 : BOOL;
		L51VA_L1 : BOOL;
		P51VB_L1 : BOOL;
		T51VB_L1 : BOOL;
		R51VB_L1 : BOOL;
		L51VB_L1 : BOOL;
		P51VC_L1 : BOOL;
		T51VC_L1 : BOOL;
		R51VC_L1 : BOOL;
		L51VC_L1 : BOOL;
		P51PA_L1 : BOOL;
		T51PA_L1 : BOOL;
		R51PA_L1 : BOOL;
		L51PA_L1 : BOOL;
		P51PB_L1 : BOOL;
		T51PB_L1 : BOOL;
		R51PB_L1 : BOOL;
		L51PB_L1 : BOOL;
		P51PC_L1 : BOOL;
		T51PC_L1 : BOOL;
		R51PC_L1 : BOOL;
		L51PC_L1 : BOOL;
		P51Q_L1 : BOOL;
		T51Q_L1 : BOOL;
		R51Q_L1 : BOOL;
		L51Q_L1 : BOOL;
		P51G_L1 : BOOL;
		T51G_L1 : BOOL;
		R51G_L1 : BOOL;
		L51G_L1 : BOOL;
		P24_L1 : BOOL;
		T24_L1 : BOOL;
		L24_L1 : BOOL;
		P40_L1 : BOOL;
		T40_L1 : BOOL;
		L40_L1 : BOOL;
		P40_L2 : BOOL;
		T40_L2 : BOOL;
		L40_L2 : BOOL;
		RpmFault : BOOL;
		var1 : BOOL;
		var2 : BOOL;
		var3 : BOOL;
		var4 : BOOL;
		var5 : BOOL;
		var6 : BOOL;
		var7 : BOOL;
		var8 : BOOL;
		var9 : BOOL;
		var10 : BOOL;
		var11 : BOOL;
		var12 : BOOL;
		var13 : BOOL;
		var14 : BOOL;
		var15 : BOOL;
		var16 : BOOL;
		var17 : BOOL;
		var18 : BOOL;
		var19 : BOOL;
		var20 : BOOL;
		var21 : BOOL;
		var22 : BOOL;
		var23 : BOOL;
		var24 : BOOL;
		var25 : BOOL;
		var26 : BOOL;
		var27 : BOOL;
		var28 : BOOL;
		var29 : BOOL;
		var30 : BOOL;
		var31 : BOOL;
		var32 : BOOL;
	END_STRUCT;
END_TYPE
```

### Local.var
```iecst
(*Protection 59*)
VAR
	P59A_L1 : PgsProt62;
	P59B_L1 : PgsProt62;
	P59C_L1 : PgsProt62;
	P59AB_L1 : PgsProt62;
	P59BC_L1 : PgsProt62;
	P59CA_L1 : PgsProt62;
	P59V1_L1 : PgsProt62;
	P59Q_L1 : PgsProt62;
	P59G_L1 : PgsProt62;
	P59A_L2 : PgsProt62;
	P59B_L2 : PgsProt62;
	P59C_L2 : PgsProt62;
	P59AB_L2 : PgsProt62;
	P59BC_L2 : PgsProt62;
	P59CA_L2 : PgsProt62;
	P59V1_L2 : PgsProt62;
	P59Q_L2 : PgsProt62;
	P59G_L2 : PgsProt62;
END_VAR
(*Protection 27*)
VAR
	P27A_L1 : PgsProt62;
	P27B_L1 : PgsProt62;
	P27C_L1 : PgsProt62;
	P27AB_L1 : PgsProt62;
	P27BC_L1 : PgsProt62;
	P27CA_L1 : PgsProt62;
	P27V1_L1 : PgsProt62;
	P27A_L2 : PgsProt62;
	P27B_L2 : PgsProt62;
	P27C_L2 : PgsProt62;
	P27AB_L2 : PgsProt62;
	P27BC_L2 : PgsProt62;
	P27CA_L2 : PgsProt62;
	P27V1_L2 : PgsProt62;
END_VAR
(*Protection 81*)
VAR
	P81O_L1 : PgsProt62;
	P81O_L2 : PgsProt62;
	P81U_L1 : PgsProt62;
	P81U_L2 : PgsProt62;
END_VAR
(*Protection 32*)
VAR
	P32OP_L1 : PgsProt62;
	P32UP_L1 : PgsProt62;
	P32OQ_L1 : PgsProt62;
	P32UQ_L1 : PgsProt62;
END_VAR
(*Protection 24*)
VAR
	P24_L1 : PgsProt24;
END_VAR
(*Protection 40*)
VAR
	P40_L1 : PgsProt40;
	P40_L2 : PgsProt40;
END_VAR
(*Protection 50*)
VAR
	P50PA_L1 : PgsProt62;
	P50PB_L1 : PgsProt62;
	P50PC_L1 : PgsProt62;
	P50Q_L1 : PgsProt62;
	P50G_L1 : PgsProt62;
	P50PA_L2 : PgsProt62;
	P50PB_L2 : PgsProt62;
	P50PC_L2 : PgsProt62;
	P50Q_L2 : PgsProt62;
	P50G_L2 : PgsProt62;
END_VAR
(*Protection 51*)
VAR
	P51VA_L1 : PgsProt51V;
	P51VB_L1 : PgsProt51V;
	P51VC_L1 : PgsProt51V;
	P51PA_L1 : PgsProt51V;
	P51PB_L1 : PgsProt51V;
	P51PC_L1 : PgsProt51V;
	P51Q_L1 : PgsProt51V;
	P51G_L1 : PgsProt51V;
END_VAR
(*Insert your comment here.*)
VAR
	P50BF : PgsProt50BF;
END_VAR
```

### Program Logical/Kontrol/Protection/Protection (IEC)
